(* PLC project robot6axis_ctrled, Dassault Systèmes ControlBuild 2021x HF2 *)
(* stored: creationDateTime 2021-06-01T17:00:16-01:00 *)

CONFIGURATION robot6axis_ctrled
  VAR_GLOBAL
    armOrigin AT 17 : ARRAY[1..3] OF REAL := [800.0, 400.0, 0.0];
    profileNr AT 523 : DINT := 0;
    HomeCmd AT 5 : BOOL := false;
    MoveVelCmd AT 6 : BOOL := false;
    MoveAbsCmd AT 7 : BOOL := false;
    MoveVel1ManualCmd AT 8 : BOOL := false;
    MoveVel2ManualCmd AT 9 : BOOL := false;
    MoveAbs1ManualCmd AT 10 : BOOL := false;
    MoveAbs2ManualCmd AT 11 : BOOL := false;
    StopCmd AT 12 : BOOL := false;
    MovePosition AT 22 : REAL := 0.0;
    MoveSpeed AT 23 : REAL := 100.0;
    MoveAcceleration AT 24 : REAL := 100.0;
    MoveDeceleration AT 25 : REAL := 100.0;
    offsetAxToMa AT 26 : REAL := 0.0;
    gripSyringes AT 13 : BOOL := false;
    Auto AT 14 : BOOL := false;
    Manu AT 15 : BOOL := false;
    run AT 16 : BOOL := false;
    armExtrem AT 27 : ARRAY[1..3] OF REAL := [3(0.0)];
    velX AT 32 : REAL := 0.0;
    velY AT 33 : REAL := 0.0;
    velZ AT 34 : REAL := 0.0;
    armInStop AT 17 : BOOL := false;
    masterPosition AT 35 : REAL := 0.0;
    ActualPositionAx AT 36 : REAL := 0.0;
    robot6axis_cams/profileNr AT 523 : DINT := 0;
    robot6axis_cams/HomeCmd AT 5 : BOOL := false;
    robot6axis_cams/MoveVelCmd AT 6 : BOOL := false;
    robot6axis_cams/MoveAbsCmd AT 7 : BOOL := false;
    robot6axis_cams/MoveVel1ManualCmd AT 8 : BOOL := false;
    robot6axis_cams/MoveVel2ManualCmd AT 9 : BOOL := false;
    robot6axis_cams/MoveAbs1ManualCmd AT 10 : BOOL := false;
    robot6axis_cams/MoveAbs2ManualCmd AT 11 : BOOL := false;
    robot6axis_cams/StopCmd AT 12 : BOOL := false;
    robot6axis_cams/MovePosition AT 22 : REAL := 0.0;
    robot6axis_cams/MoveSpeed AT 23 : REAL := 100.0;
    robot6axis_cams/MoveAcceleration AT 24 : REAL := 100.0;
    robot6axis_cams/MoveDeceleration AT 25 : REAL := 100.0;
    robot6axis_cams/offsetAxToMa AT 26 : REAL := 0.0;
    robot6axis_cams/name1 AT 636 : STRING(50) := 'CamAxis1_100.txt';
    robot6axis_cams/name2 AT 583 : STRING(50) := 'CamAxis2_100.txt';
    robot6axis_cams/name3 AT 530 : STRING(50) := 'CamAxis3_100.txt';
    robot6axis_cams/name4 AT 477 : STRING(50) := 'CamAxis4_100.txt';
    robot6axis_cams/name5 AT 424 : STRING(50) := 'CamAxis5_100.txt';
    robot6axis_cams/name6 AT 371 : STRING(50) := 'CamAxis6_100.txt';
    robot6axis_cams/name1_rej AT 318 : STRING(50) := 'CamAxis1_rej.txt';
    robot6axis_cams/name2_rej AT 265 : STRING(50) := 'CamAxis2_rej.txt';
    robot6axis_cams/name3_rej AT 212 : STRING(50) := 'CamAxis3_rej.txt';
    robot6axis_cams/name4_rej AT 159 : STRING(50) := 'CamAxis4_rej.txt';
    robot6axis_cams/name5_rej AT 106 : STRING(50) := 'CamAxis5_rej.txt';
    robot6axis_cams/name6_rej AT 53 : STRING(50) := 'CamAxis6_rej.txt';
    robot6axis_cams/slavePosition1 AT 158 : REAL := 0.0;
    robot6axis_cams/slavePosition2 AT 159 : REAL := 0.0;
    robot6axis_cams/slavePosition3 AT 160 : REAL := 0.0;
    robot6axis_cams/slavePosition4 AT 161 : REAL := 0.0;
    robot6axis_cams/slavePosition5 AT 162 : REAL := 0.0;
    robot6axis_cams/slavePosition6 AT 163 : REAL := 0.0;
    robot6axis_cams/ActualPositionAx AT 36 : REAL := 0.0;
    robot6axis_cams/masterPosition AT 35 : REAL := 0.0;
    robot6axis_cams/servo_kinetix2/status AT 549 : INT := 0;
    robot6axis_cams/servo_kinetix2/errorFlag AT 548 : INT := 0;
    robot6axis_cams/servo_kinetix2/ActualPositionAx1 AT 2630 : REAL := 0.0;
    robot6axis_cams/servo_kinetix2/MoveVelDone1 AT 87 : BOOL := false;
    robot6axis_cams/servo_kinetix2/ActualVelocity1 AT 2629 : REAL := 0.0;
    robot6axis_cams/servo_kinetix2/MoveAbsDone1 AT 86 : BOOL := false;
    robot6axis_cams/servo_kinetix2/HomeCmd AT 5 : BOOL := false;
    robot6axis_cams/servo_kinetix2/MoveVelCmd AT 6 : BOOL := false;
    robot6axis_cams/servo_kinetix2/MoveAbsCmd AT 7 : BOOL := false;
    robot6axis_cams/servo_kinetix2/MoveVel1ManualCmd AT 8 : BOOL := false;
    robot6axis_cams/servo_kinetix2/MoveVel2ManualCmd AT 9 : BOOL := false;
    robot6axis_cams/servo_kinetix2/MoveAbs1ManualCmd AT 10 : BOOL := false;
    robot6axis_cams/servo_kinetix2/MoveAbs2ManualCmd AT 11 : BOOL := false;
    robot6axis_cams/servo_kinetix2/StopCmd AT 12 : BOOL := false;
    robot6axis_cams/servo_kinetix2/MovePosition AT 22 : REAL := 0.0;
    robot6axis_cams/servo_kinetix2/MoveSpeed AT 23 : REAL := 100.0;
    robot6axis_cams/servo_kinetix2/MoveAcceleration AT 24 : REAL := 100.0;
    robot6axis_cams/servo_kinetix2/MoveDeceleration AT 25 : REAL := 100.0;
    robot6axis_cams/servo_kinetix2/offsetAxToMa AT 26 : REAL := 0.0;
    robot6axis_cams/servo_kinetix2/PLC_StatusReady AT 85 : BOOL := true;
    robot6axis_cams/servo_kinetix2/PLC_StatusMoved AT 84 : BOOL := false;
    robot6axis_cams/servo_kinetix2/PLC_StatusStand AT 83 : BOOL := false;
    robot6axis_cams/servo_kinetix2/PLC_ActualPositionAx AT 2628 : REAL := 0.0;
    robot6axis_cams/servo_kinetix2/PLC_ActualPositionMa AT 2627 : REAL := 0.0;
    robot6axis_cams/servo_kinetix2/PLC_ActualVelocity AT 2626 : REAL := 0.0;
    robot6axis_cams/servo_kinetix2/physicalPosInit AT 2625 : REAL := 0.0;
    robot6axis_cams/servo_kinetix2/MAX_SPEED AT 2624 : REAL(0.0..3.4e+038) := 30.0;
    robot6axis_cams/servo_kinetix2/MAX_ACCEL AT 2623 : REAL(0.0..3.4e+038) := 1500.0;
    robot6axis_cams/servo_kinetix2/MAX_DECEL AT 2622 : REAL(0.0..3.4e+038) := 1500.0;
    robot6axis_cams/servo_kinetix2/MODULO_LENGTH AT 2621 : REAL := 0.0;
    robot6axis_cams/servo_kinetix2/StatusReady AT 82 : BOOL := true;
    robot6axis_cams/servo_kinetix2/StatusMoved AT 81 : BOOL := false;
    robot6axis_cams/servo_kinetix2/StatusStand AT 80 : BOOL := false;
    robot6axis_cams/servo_kinetix2/ActualPositionAx AT 36 : REAL := 0.0;
    robot6axis_cams/servo_kinetix2/ActualPositionMa AT 2620 : REAL := 0.0;
    robot6axis_cams/servo_kinetix2/ActualVelocity AT 2619 : REAL := 0.0;
    robot6axis_cams/servo_kinetix2/MaximumVelocity AT 2618 : REAL := 0.0;
    robot6axis_cams/servo_kinetix2/StatusPosIncrease AT 79 : BOOL := false;
    robot6axis_cams/servo_kinetix2/StatusPosDecrease AT 78 : BOOL := false;
    robot6axis_cams/servo_kinetix2/displayJauge AT 2617 : REAL := 0.0;
    robot6axis_cams/servo_kinetix2/servo_mode/PLC_StatusReady AT 85 : BOOL := true;
    robot6axis_cams/servo_kinetix2/servo_mode/PLC_StatusMoved AT 84 : BOOL := false;
    robot6axis_cams/servo_kinetix2/servo_mode/PLC_StatusStand AT 83 : BOOL := false;
    robot6axis_cams/servo_kinetix2/servo_mode/PLC_ActualPositionAx AT 2628 : REAL := 0.0;
    robot6axis_cams/servo_kinetix2/servo_mode/PLC_ActualPositionMa AT 2627 : REAL := 0.0;
    robot6axis_cams/servo_kinetix2/servo_mode/PLC_ActualVelocity AT 2626 : REAL := 0.0;
    robot6axis_cams/servo_kinetix2/servo_mode/StatusReady AT 88 : BOOL := true;
    robot6axis_cams/servo_kinetix2/servo_mode/StatusMoved AT 89 : BOOL := false;
    robot6axis_cams/servo_kinetix2/servo_mode/StatusStand AT 90 : BOOL := false;
    robot6axis_cams/servo_kinetix2/servo_mode/ActualPositionMa AT 5079 : REAL := 0.0;
    robot6axis_cams/servo_kinetix2/servo_mode/ActualVelocity AT 5080 : REAL := 0.0;
    robot6axis_cams/servo_kinetix2/servo_mode/MaximumVelocity AT 5081 : REAL := 0.0;
    robot6axis_cams/servo_kinetix2/servo_mode/physicalPosInit AT 2625 : REAL := 0.0;
    robot6axis_cams/servo_kinetix2/servo_mode/ActualPositionAx AT 2630 : REAL := 0.0;
    robot6axis_cams/servo_kinetix2/servo_mode/StatusReady_o AT 82 : BOOL := true;
    robot6axis_cams/servo_kinetix2/servo_mode/StatusMoved_o AT 81 : BOOL := false;
    robot6axis_cams/servo_kinetix2/servo_mode/StatusStand_o AT 80 : BOOL := false;
    robot6axis_cams/servo_kinetix2/servo_mode/ActualPositionAx_o AT 36 : REAL := 0.0;
    robot6axis_cams/servo_kinetix2/servo_mode/ActualPositionMa_o AT 2620 : REAL := 0.0;
    robot6axis_cams/servo_kinetix2/servo_mode/ActualVelocity_o AT 2619 : REAL := 0.0;
    robot6axis_cams/servo_kinetix2/servo_mode/MaximumVelocity_o AT 2618 : REAL := 0.0;
    robot6axis_cams/servo_kinetix2/servo_mode/StatusPosIncrease_o AT 79 : BOOL := false;
    robot6axis_cams/servo_kinetix2/servo_mode/StatusPosDecrease_o AT 78 : BOOL := false;
    robot6axis_cams/servo_kinetix2/servo_mode/displayJauge_o AT 2617 : REAL := 0.0;
    robot6axis_cams/servo_kinetix2/servo_mode/PLCMode AT 95 : BOOL := false;
    robot6axis_cams/servo_kinetix2/servo_mode/PLCMode1 AT 96 : BOOL := false;
    robot6axis_cams/servo_kinetix2/servo_mode/initDone AT 97 : BOOL := false;
    robot6axis_cams/servo_kinetix2/servo_mode/displayPosMin AT 5084 : REAL := 0.0;
    robot6axis_cams/servo_kinetix2/servo_mode/displayPosMax AT 5085 : REAL := 0.0;
    robot6axis_cams/servo_kinetix2/servo_mode/PLC_ActualPositionAx1 AT 5086 : REAL := 0.0;
    robot6axis_cams/servo_kinetix2/servo_mode/PLC_ActualVelocity1 AT 5087 : REAL := 0.0;
    robot6axis_cams/servo_kinetix2/servo_mode/ActualPositionAx1 AT 5088 : REAL := 0.0;
    robot6axis_cams/servo_kinetix2/servo_mode/ActualVelocity1 AT 5089 : REAL := 0.0;
    robot6axis_cams/servo_kinetix2/servo_mode/offsetAxToMa AT 5090 : REAL := 0.0;
    robot6axis_cams/servo_kinetix2/servo_mode/offsetAxToMa1 AT 5091 : REAL := 0.0;
    robot6axis_cams/servo_kinetix2/servo_mode/ActualPositionMa_o1 AT 5092 : REAL := 0.0;
    robot6axis_cams/servo_kinetix2/servo_control/HomeCmd AT 5 : BOOL := false;
    robot6axis_cams/servo_kinetix2/servo_control/MoveVelCmd AT 6 : BOOL := false;
    robot6axis_cams/servo_kinetix2/servo_control/MoveAbsCmd AT 7 : BOOL := false;
    robot6axis_cams/servo_kinetix2/servo_control/MoveVel1ManualCmd AT 8 : BOOL := false;
    robot6axis_cams/servo_kinetix2/servo_control/MoveVel2ManualCmd AT 9 : BOOL := false;
    robot6axis_cams/servo_kinetix2/servo_control/MoveAbs1ManualCmd AT 10 : BOOL := false;
    robot6axis_cams/servo_kinetix2/servo_control/MoveAbs2ManualCmd AT 11 : BOOL := false;
    robot6axis_cams/servo_kinetix2/servo_control/StopCmd AT 12 : BOOL := false;
    robot6axis_cams/servo_kinetix2/servo_control/MovePosition AT 22 : REAL := 0.0;
    robot6axis_cams/servo_kinetix2/servo_control/MoveSpeed AT 23 : REAL := 100.0;
    robot6axis_cams/servo_kinetix2/servo_control/MoveAcceleration AT 24 : REAL := 100.0;
    robot6axis_cams/servo_kinetix2/servo_control/MoveDeceleration AT 25 : REAL := 100.0;
    robot6axis_cams/servo_kinetix2/servo_control/offsetAxToMa AT 26 : REAL := 0.0;
    robot6axis_cams/servo_kinetix2/servo_control/physicalPosInit AT 2625 : REAL := 0.0;
    robot6axis_cams/servo_kinetix2/servo_control/MAX_SPEED AT 2624 : REAL(0.0..3.4e+038) := 30.0;
    robot6axis_cams/servo_kinetix2/servo_control/status AT 549 : INT := 0;
    robot6axis_cams/servo_kinetix2/servo_control/errorFlag AT 548 : INT := 0;
    robot6axis_cams/servo_kinetix2/servo_control/IOActualPositionAx AT 2630 : REAL := 0.0;
    robot6axis_cams/servo_kinetix2/servo_control/IOVelDone AT 87 : BOOL := false;
    robot6axis_cams/servo_kinetix2/servo_control/IOAbsDone AT 86 : BOOL := false;
    robot6axis_cams/servo_kinetix2/servo_control/IOActualVelocity AT 2629 : REAL := 0.0;
    robot6axis_cams/servo_kinetix2/servo_control/OperationMode AT 574 : INT := 0;
    robot6axis_cams/servo_kinetix2/servo_control/StatusReady AT 88 : BOOL := true;
    robot6axis_cams/servo_kinetix2/servo_control/StatusMove AT 89 : BOOL := false;
    robot6axis_cams/servo_kinetix2/servo_control/StatusStand AT 90 : BOOL := false;
    robot6axis_cams/servo_kinetix2/servo_control/ActualPositionMa AT 5079 : REAL := 0.0;
    robot6axis_cams/servo_kinetix2/servo_control/ActualVelocity AT 5080 : REAL := 0.0;
    robot6axis_cams/servo_kinetix2/servo_control/MaximumVelocity AT 5081 : REAL := 0.0;
    robot6axis_cams/servo_kinetix2/servo_control/VelEnabled AT 91 : BOOL := false;
    robot6axis_cams/servo_kinetix2/servo_control/VelCmd AT 92 : BOOL := false;
    robot6axis_cams/servo_kinetix2/servo_control/PosEnabled AT 93 : BOOL := false;
    robot6axis_cams/servo_kinetix2/servo_control/PosCmd AT 94 : BOOL := false;
    robot6axis_cams/servo_kinetix2/servo_control/Position AT 5083 : REAL := 0.0;
    robot6axis_cams/servo_kinetix2/servo_control/Speed AT 5082 : REAL := 0.0;
    robot6axis_cams/servo_kinetix2/servo_control/ManualMode AT 575 : INT := 0;
    robot6axis_cams/servo_kinetix2/servo_control/initDone AT 98 : BOOL := false;
    robot6axis_cams/servo_kinetix2/servo_control/ActualPositionMa1 AT 5093 : REAL := 0.0;
    robot6axis_cams/servo_kinetix2/servo_control/offsetAxToMa1 AT 5094 : REAL := 0.0;
    robot6axis_cams/servo_kinetix2/servo_control/HOME_POSITION AT 5095 : REAL := 100.0;
    robot6axis_cams/servo_kinetix2/servo_control/MANUAL_POSITION1 AT 5096 : REAL := 0.0;
    robot6axis_cams/servo_kinetix2/servo_control/MANUAL_POSITION2 AT 5097 : REAL := 150.0;
    robot6axis_cams/servo_kinetix2/servo_control/MANUAL_SPEED1 AT 5098 : REAL := -100.0;
    robot6axis_cams/servo_kinetix2/servo_control/MANUAL_SPEED2 AT 5099 : REAL := 100.0;
    robot6axis_cams/servo_kinetix2/servo_control/MANUAL_SPEED AT 5100 : REAL := 100.0;
    robot6axis_cams/servo_kinetix2/servo_velocity/MoveVelEnable AT 91 : BOOL := false;
    robot6axis_cams/servo_kinetix2/servo_velocity/MoveVelStart AT 92 : BOOL := false;
    robot6axis_cams/servo_kinetix2/servo_velocity/MoveSpeed AT 5082 : REAL := 0.0;
    robot6axis_cams/servo_kinetix2/servo_velocity/MoveAcceleration AT 24 : REAL := 100.0;
    robot6axis_cams/servo_kinetix2/servo_velocity/MoveDeceleration AT 25 : REAL := 100.0;
    robot6axis_cams/servo_kinetix2/servo_velocity/MAX_SPEED AT 2624 : REAL(0.0..3.4e+038) := 30.0;
    robot6axis_cams/servo_kinetix2/servo_velocity/MAX_ACCEL AT 2623 : REAL(0.0..3.4e+038) := 1500.0;
    robot6axis_cams/servo_kinetix2/servo_velocity/MAX_DECEL AT 2622 : REAL(0.0..3.4e+038) := 1500.0;
    robot6axis_cams/servo_kinetix2/servo_velocity/MODULO_LENGTH AT 2621 : REAL := 0.0;
    robot6axis_cams/servo_kinetix2/servo_velocity/status AT 549 : INT := 0;
    robot6axis_cams/servo_kinetix2/servo_velocity/errorFlag AT 548 : INT := 0;
    robot6axis_cams/servo_kinetix2/servo_velocity/MoveVelDone AT 87 : BOOL := false;
    robot6axis_cams/servo_kinetix2/servo_velocity/ActualPositionAx AT 2630 : REAL := 0.0;
    robot6axis_cams/servo_kinetix2/servo_velocity/ActualVelocity AT 2629 : REAL := 0.0;
    robot6axis_cams/servo_kinetix2/servo_velocity/firstStep AT 99 : BOOL := true;
    robot6axis_cams/servo_kinetix2/servo_velocity/stepDone AT 100 : BOOL := false;
    robot6axis_cams/servo_kinetix2/servo_velocity/currentTime AT 5101 : REAL := 0.0;
    robot6axis_cams/servo_kinetix2/servo_velocity/MoveSpeed1 AT 5102 : REAL := 0.0;
    robot6axis_cams/servo_kinetix2/servo_velocity/acceleration AT 5103 : REAL := 0.0;
    robot6axis_cams/servo_kinetix2/servo_velocity/deceleration AT 5104 : REAL := 0.0;
    robot6axis_cams/servo_kinetix2/servo_velocity/orderSpeed AT 5105 : REAL := 0.0;
    robot6axis_cams/servo_kinetix2/servo_velocity/endChangeSpeed AT 5106 : REAL := 0.0;
    robot6axis_cams/servo_kinetix2/servo_velocity/accelDecelChangeSpeed AT 5107 : REAL := 0.0;
    robot6axis_cams/servo_kinetix2/servo_velocity/ActualVelocity1 AT 5108 : REAL := 0.0;
    robot6axis_cams/servo_kinetix2/servo_velocity/speedChanged AT 101 : BOOL := false;
    robot6axis_cams/servo_kinetix2/servo_position/MoveAbsEnable AT 93 : BOOL := false;
    robot6axis_cams/servo_kinetix2/servo_position/MoveAbsStart AT 94 : BOOL := false;
    robot6axis_cams/servo_kinetix2/servo_position/MovePosition AT 5083 : REAL := 0.0;
    robot6axis_cams/servo_kinetix2/servo_position/MoveSpeed AT 5082 : REAL := 0.0;
    robot6axis_cams/servo_kinetix2/servo_position/MoveAcceleration AT 24 : REAL := 100.0;
    robot6axis_cams/servo_kinetix2/servo_position/MoveDeceleration AT 25 : REAL := 100.0;
    robot6axis_cams/servo_kinetix2/servo_position/MAX_SPEED AT 2624 : REAL(0.0..3.4e+038) := 30.0;
    robot6axis_cams/servo_kinetix2/servo_position/MAX_ACCEL AT 2623 : REAL(0.0..3.4e+038) := 1500.0;
    robot6axis_cams/servo_kinetix2/servo_position/MAX_DECEL AT 2622 : REAL(0.0..3.4e+038) := 1500.0;
    robot6axis_cams/servo_kinetix2/servo_position/MODULO_LENGTH AT 2621 : REAL := 0.0;
    robot6axis_cams/servo_kinetix2/servo_position/status AT 549 : INT := 0;
    robot6axis_cams/servo_kinetix2/servo_position/errorFlag AT 548 : INT := 0;
    robot6axis_cams/servo_kinetix2/servo_position/MoveAbsDone AT 86 : BOOL := false;
    robot6axis_cams/servo_kinetix2/servo_position/ActualPositionAx AT 2630 : REAL := 0.0;
    robot6axis_cams/servo_kinetix2/servo_position/ActualVelocity AT 2629 : REAL := 0.0;
    robot6axis_cams/servo_kinetix2/servo_position/firstStep AT 102 : BOOL := true;
    robot6axis_cams/servo_kinetix2/servo_position/stepDone AT 103 : BOOL := false;
    robot6axis_cams/servo_kinetix2/servo_position/timeToStop AT 5109 : REAL := 0.0;
    robot6axis_cams/servo_kinetix2/servo_position/distanceToStop AT 5110 : REAL := 0.0;
    robot6axis_cams/servo_kinetix2/servo_position/distance AT 5111 : REAL := 0.0;
    robot6axis_cams/servo_kinetix2/servo_position/currentTime AT 5112 : REAL := 0.0;
    robot6axis_cams/servo_kinetix2/servo_position/currentSpeed1 AT 5113 : REAL := 0.0;
    robot6axis_cams/servo_kinetix2/servo_position/targetPosition AT 5114 : REAL := 0.0;
    robot6axis_cams/servo_kinetix2/servo_position/ActualPositionAx1 AT 5115 : REAL := 0.0;
    robot6axis_cams/servo_kinetix2/servo_position/acceleration AT 5116 : REAL := 0.0;
    robot6axis_cams/servo_kinetix2/servo_position/deceleration AT 5117 : REAL := 0.0;
    robot6axis_cams/servo_kinetix2/servo_position/orderSpeed AT 5118 : REAL := 0.0;
    robot6axis_cams/servo_kinetix2/servo_position/moveDirection AT 5119 : REAL := 0.0;
    robot6axis_cams/servo_kinetix2/servo_position/moveDirection1 AT 5120 : REAL := 0.0;
    robot6axis_cams/servo_kinetix2/servo_position/endChangeSpeed AT 5121 : REAL := 0.0;
    robot6axis_cams/servo_kinetix2/servo_position/ActualVelocity1 AT 5122 : REAL := 0.0;
    robot6axis_cams/cam_profile1/name AT 636 : STRING(50) := 'CamAxis1_100.txt';
    robot6axis_cams/cam_profile1/nbPoints AT 550 : INT := 0;
    robot6axis_cams/cam_profile1/MasterPoints AT 2631 : ARRAY[1..100] OF REAL := [100(0.0)];
    robot6axis_cams/cam_profile1/SlavePoints AT 2733 : ARRAY[1..100] OF REAL := [100(0.0)];
    robot6axis_cams/cam_profile1/pointer AT 551 : DINT := 0;
    robot6axis_cams/cam_profile1/initialized AT 104 : BOOL := false;
    robot6axis_cams/cam_profile1/pFile AT 576 : DINT := 0;
    robot6axis_cams/cam_profile1/fault_reading AT 105 : BOOL := false;
    robot6axis_cams/cam_profile1/fault_openning AT 106 : BOOL := false;
    robot6axis_cams/cam_profile1/complete_path AT 689 : STRING(254) := '';
    robot6axis_cams/cam_profile7/name AT 318 : STRING(50) := 'CamAxis1_rej.txt';
    robot6axis_cams/cam_profile7/nbPoints AT 552 : INT := 0;
    robot6axis_cams/cam_profile7/MasterPoints AT 2835 : ARRAY[1..100] OF REAL := [100(0.0)];
    robot6axis_cams/cam_profile7/SlavePoints AT 2937 : ARRAY[1..100] OF REAL := [100(0.0)];
    robot6axis_cams/cam_profile7/pointer AT 553 : DINT := 0;
    robot6axis_cams/cam_profile7/initialized AT 107 : BOOL := false;
    robot6axis_cams/cam_profile7/pFile AT 577 : DINT := 0;
    robot6axis_cams/cam_profile7/fault_reading AT 108 : BOOL := false;
    robot6axis_cams/cam_profile7/fault_openning AT 109 : BOOL := false;
    robot6axis_cams/cam_profile7/complete_path AT 946 : STRING(254) := '';
    robot6axis_cams/cam_computation1/profileNr AT 523 : DINT := 0;
    robot6axis_cams/cam_computation1/MasterPositionIn AT 36 : REAL := 0.0;
    robot6axis_cams/cam_computation1/nbPoints0 AT 550 : INT := 0;
    robot6axis_cams/cam_computation1/MasterPoints0 AT 2631 : ARRAY[1..100] OF REAL := [100(0.0)];
    robot6axis_cams/cam_computation1/SlavePoints0 AT 2733 : ARRAY[1..100] OF REAL := [100(0.0)];
    robot6axis_cams/cam_computation1/pointer0 AT 551 : DINT := 0;
    robot6axis_cams/cam_computation1/nbPoints1 AT 552 : INT := 0;
    robot6axis_cams/cam_computation1/MasterPoints1 AT 2835 : ARRAY[1..100] OF REAL := [100(0.0)];
    robot6axis_cams/cam_computation1/SlavePoints1 AT 2937 : ARRAY[1..100] OF REAL := [100(0.0)];
    robot6axis_cams/cam_computation1/pointer1 AT 553 : DINT := 0;
    robot6axis_cams/cam_computation1/nbPoints2 AT 547 : INT := 0;
    robot6axis_cams/cam_computation1/MasterPoints2 AT 2515 : ARRAY[1..100] OF REAL := [100(0.0)];
    robot6axis_cams/cam_computation1/SlavePoints2 AT 2413 : ARRAY[1..100] OF REAL := [100(0.0)];
    robot6axis_cams/cam_computation1/pointer2 AT 546 : DINT := 0;
    robot6axis_cams/cam_computation1/nbPoints3 AT 545 : INT := 0;
    robot6axis_cams/cam_computation1/MasterPoints3 AT 2311 : ARRAY[1..100] OF REAL := [100(0.0)];
    robot6axis_cams/cam_computation1/SlavePoints3 AT 2209 : ARRAY[1..100] OF REAL := [100(0.0)];
    robot6axis_cams/cam_computation1/pointer3 AT 544 : DINT := 0;
    robot6axis_cams/cam_computation1/slavePosition AT 158 : REAL := 0.0;
    robot6axis_cams/cam_computation1/masterPosition AT 35 : REAL := 0.0;
    robot6axis_cams/cam_computation1/i AT 578 : INT := 0;
    robot6axis_cams/cam_computation1/modulo AT 5123 : REAL := 0.0;
    robot6axis_cams/cam_computation1/divider AT 579 : INT := 0;
    robot6axis_cams/cam_computation1/faultProfileNr AT 110 : BOOL := false;
    robot6axis_cams/cam_computation1/faultMasterPositionOOB AT 111 : BOOL := false;
    robot6axis_cams/cam_computation1/faultLinComputation AT 112 : BOOL := false;
    robot6axis_cams/cam_computation1/nbPoints AT 580 : INT := 0;
    robot6axis_cams/cam_computation1/MasterPoints AT 5124 : ARRAY[1..100] OF REAL := [100(0.0)];
    robot6axis_cams/cam_computation1/SlavePoints AT 5226 : ARRAY[1..100] OF REAL := [100(0.0)];
    robot6axis_cams/cam_computation1/found AT 113 : BOOL := false;
    robot6axis_cams/cam_computation1/index AT 581 : INT := 0;
    robot6axis_cams/cam_computation1/linDenom AT 5328 : REAL := 0.0;
    robot6axis_cams/cam_computation1/linNum AT 5329 : REAL := 0.0;
    robot6axis_cams/cam_computation1/linA AT 5330 : REAL := 0.0;
    robot6axis_cams/cam_computation1/linB AT 5331 : REAL := 0.0;
    robot6axis_cams/cam_computation1/FACTOR AT 5332 : REAL := 1.0;
    robot6axis_cams/cam_profile2/name AT 583 : STRING(50) := 'CamAxis2_100.txt';
    robot6axis_cams/cam_profile2/nbPoints AT 554 : INT := 0;
    robot6axis_cams/cam_profile2/MasterPoints AT 3039 : ARRAY[1..100] OF REAL := [100(0.0)];
    robot6axis_cams/cam_profile2/SlavePoints AT 3141 : ARRAY[1..100] OF REAL := [100(0.0)];
    robot6axis_cams/cam_profile2/pointer AT 555 : DINT := 0;
    robot6axis_cams/cam_profile2/initialized AT 114 : BOOL := false;
    robot6axis_cams/cam_profile2/pFile AT 582 : DINT := 0;
    robot6axis_cams/cam_profile2/fault_reading AT 115 : BOOL := false;
    robot6axis_cams/cam_profile2/fault_openning AT 116 : BOOL := false;
    robot6axis_cams/cam_profile2/complete_path AT 1203 : STRING(254) := '';
    robot6axis_cams/cam_profile8/name AT 265 : STRING(50) := 'CamAxis2_rej.txt';
    robot6axis_cams/cam_profile8/nbPoints AT 556 : INT := 0;
    robot6axis_cams/cam_profile8/MasterPoints AT 3243 : ARRAY[1..100] OF REAL := [100(0.0)];
    robot6axis_cams/cam_profile8/SlavePoints AT 3345 : ARRAY[1..100] OF REAL := [100(0.0)];
    robot6axis_cams/cam_profile8/pointer AT 557 : DINT := 0;
    robot6axis_cams/cam_profile8/initialized AT 117 : BOOL := false;
    robot6axis_cams/cam_profile8/pFile AT 583 : DINT := 0;
    robot6axis_cams/cam_profile8/fault_reading AT 118 : BOOL := false;
    robot6axis_cams/cam_profile8/fault_openning AT 119 : BOOL := false;
    robot6axis_cams/cam_profile8/complete_path AT 1460 : STRING(254) := '';
    robot6axis_cams/cam_computation2/profileNr AT 523 : DINT := 0;
    robot6axis_cams/cam_computation2/MasterPositionIn AT 36 : REAL := 0.0;
    robot6axis_cams/cam_computation2/nbPoints0 AT 554 : INT := 0;
    robot6axis_cams/cam_computation2/MasterPoints0 AT 3039 : ARRAY[1..100] OF REAL := [100(0.0)];
    robot6axis_cams/cam_computation2/SlavePoints0 AT 3141 : ARRAY[1..100] OF REAL := [100(0.0)];
    robot6axis_cams/cam_computation2/pointer0 AT 555 : DINT := 0;
    robot6axis_cams/cam_computation2/nbPoints1 AT 556 : INT := 0;
    robot6axis_cams/cam_computation2/MasterPoints1 AT 3243 : ARRAY[1..100] OF REAL := [100(0.0)];
    robot6axis_cams/cam_computation2/SlavePoints1 AT 3345 : ARRAY[1..100] OF REAL := [100(0.0)];
    robot6axis_cams/cam_computation2/pointer1 AT 557 : DINT := 0;
    robot6axis_cams/cam_computation2/nbPoints2 AT 543 : INT := 0;
    robot6axis_cams/cam_computation2/MasterPoints2 AT 2107 : ARRAY[1..100] OF REAL := [100(0.0)];
    robot6axis_cams/cam_computation2/SlavePoints2 AT 2005 : ARRAY[1..100] OF REAL := [100(0.0)];
    robot6axis_cams/cam_computation2/pointer2 AT 542 : DINT := 0;
    robot6axis_cams/cam_computation2/nbPoints3 AT 541 : INT := 0;
    robot6axis_cams/cam_computation2/MasterPoints3 AT 1903 : ARRAY[1..100] OF REAL := [100(0.0)];
    robot6axis_cams/cam_computation2/SlavePoints3 AT 1801 : ARRAY[1..100] OF REAL := [100(0.0)];
    robot6axis_cams/cam_computation2/pointer3 AT 540 : DINT := 0;
    robot6axis_cams/cam_computation2/slavePosition AT 159 : REAL := 0.0;
    robot6axis_cams/cam_computation2/masterPosition AT 1800 : REAL := 0.0;
    robot6axis_cams/cam_computation2/i AT 584 : INT := 0;
    robot6axis_cams/cam_computation2/modulo AT 5333 : REAL := 0.0;
    robot6axis_cams/cam_computation2/divider AT 585 : INT := 0;
    robot6axis_cams/cam_computation2/faultProfileNr AT 120 : BOOL := false;
    robot6axis_cams/cam_computation2/faultMasterPositionOOB AT 121 : BOOL := false;
    robot6axis_cams/cam_computation2/faultLinComputation AT 122 : BOOL := false;
    robot6axis_cams/cam_computation2/nbPoints AT 586 : INT := 0;
    robot6axis_cams/cam_computation2/MasterPoints AT 5334 : ARRAY[1..100] OF REAL := [100(0.0)];
    robot6axis_cams/cam_computation2/SlavePoints AT 5436 : ARRAY[1..100] OF REAL := [100(0.0)];
    robot6axis_cams/cam_computation2/found AT 123 : BOOL := false;
    robot6axis_cams/cam_computation2/index AT 587 : INT := 0;
    robot6axis_cams/cam_computation2/linDenom AT 5538 : REAL := 0.0;
    robot6axis_cams/cam_computation2/linNum AT 5539 : REAL := 0.0;
    robot6axis_cams/cam_computation2/linA AT 5540 : REAL := 0.0;
    robot6axis_cams/cam_computation2/linB AT 5541 : REAL := 0.0;
    robot6axis_cams/cam_computation2/FACTOR AT 5542 : REAL := 1.0;
    robot6axis_cams/cam_profile3/name AT 530 : STRING(50) := 'CamAxis3_100.txt';
    robot6axis_cams/cam_profile3/nbPoints AT 558 : INT := 0;
    robot6axis_cams/cam_profile3/MasterPoints AT 3447 : ARRAY[1..100] OF REAL := [100(0.0)];
    robot6axis_cams/cam_profile3/SlavePoints AT 3549 : ARRAY[1..100] OF REAL := [100(0.0)];
    robot6axis_cams/cam_profile3/pointer AT 559 : DINT := 0;
    robot6axis_cams/cam_profile3/initialized AT 124 : BOOL := false;
    robot6axis_cams/cam_profile3/pFile AT 588 : DINT := 0;
    robot6axis_cams/cam_profile3/fault_reading AT 125 : BOOL := false;
    robot6axis_cams/cam_profile3/fault_openning AT 126 : BOOL := false;
    robot6axis_cams/cam_profile3/complete_path AT 1717 : STRING(254) := '';
    robot6axis_cams/cam_profile9/name AT 212 : STRING(50) := 'CamAxis3_rej.txt';
    robot6axis_cams/cam_profile9/nbPoints AT 560 : INT := 0;
    robot6axis_cams/cam_profile9/MasterPoints AT 3651 : ARRAY[1..100] OF REAL := [100(0.0)];
    robot6axis_cams/cam_profile9/SlavePoints AT 3753 : ARRAY[1..100] OF REAL := [100(0.0)];
    robot6axis_cams/cam_profile9/pointer AT 561 : DINT := 0;
    robot6axis_cams/cam_profile9/initialized AT 127 : BOOL := false;
    robot6axis_cams/cam_profile9/pFile AT 589 : DINT := 0;
    robot6axis_cams/cam_profile9/fault_reading AT 128 : BOOL := false;
    robot6axis_cams/cam_profile9/fault_openning AT 129 : BOOL := false;
    robot6axis_cams/cam_profile9/complete_path AT 1974 : STRING(254) := '';
    robot6axis_cams/cam_computation3/profileNr AT 523 : DINT := 0;
    robot6axis_cams/cam_computation3/MasterPositionIn AT 36 : REAL := 0.0;
    robot6axis_cams/cam_computation3/nbPoints0 AT 558 : INT := 0;
    robot6axis_cams/cam_computation3/MasterPoints0 AT 3447 : ARRAY[1..100] OF REAL := [100(0.0)];
    robot6axis_cams/cam_computation3/SlavePoints0 AT 3549 : ARRAY[1..100] OF REAL := [100(0.0)];
    robot6axis_cams/cam_computation3/pointer0 AT 559 : DINT := 0;
    robot6axis_cams/cam_computation3/nbPoints1 AT 560 : INT := 0;
    robot6axis_cams/cam_computation3/MasterPoints1 AT 3651 : ARRAY[1..100] OF REAL := [100(0.0)];
    robot6axis_cams/cam_computation3/SlavePoints1 AT 3753 : ARRAY[1..100] OF REAL := [100(0.0)];
    robot6axis_cams/cam_computation3/pointer1 AT 561 : DINT := 0;
    robot6axis_cams/cam_computation3/nbPoints2 AT 539 : INT := 0;
    robot6axis_cams/cam_computation3/MasterPoints2 AT 1698 : ARRAY[1..100] OF REAL := [100(0.0)];
    robot6axis_cams/cam_computation3/SlavePoints2 AT 1596 : ARRAY[1..100] OF REAL := [100(0.0)];
    robot6axis_cams/cam_computation3/pointer2 AT 538 : DINT := 0;
    robot6axis_cams/cam_computation3/nbPoints3 AT 537 : INT := 0;
    robot6axis_cams/cam_computation3/MasterPoints3 AT 1494 : ARRAY[1..100] OF REAL := [100(0.0)];
    robot6axis_cams/cam_computation3/SlavePoints3 AT 1392 : ARRAY[1..100] OF REAL := [100(0.0)];
    robot6axis_cams/cam_computation3/pointer3 AT 536 : DINT := 0;
    robot6axis_cams/cam_computation3/slavePosition AT 160 : REAL := 0.0;
    robot6axis_cams/cam_computation3/masterPosition AT 1391 : REAL := 0.0;
    robot6axis_cams/cam_computation3/i AT 590 : INT := 0;
    robot6axis_cams/cam_computation3/modulo AT 5543 : REAL := 0.0;
    robot6axis_cams/cam_computation3/divider AT 591 : INT := 0;
    robot6axis_cams/cam_computation3/faultProfileNr AT 130 : BOOL := false;
    robot6axis_cams/cam_computation3/faultMasterPositionOOB AT 131 : BOOL := false;
    robot6axis_cams/cam_computation3/faultLinComputation AT 132 : BOOL := false;
    robot6axis_cams/cam_computation3/nbPoints AT 592 : INT := 0;
    robot6axis_cams/cam_computation3/MasterPoints AT 5544 : ARRAY[1..100] OF REAL := [100(0.0)];
    robot6axis_cams/cam_computation3/SlavePoints AT 5646 : ARRAY[1..100] OF REAL := [100(0.0)];
    robot6axis_cams/cam_computation3/found AT 133 : BOOL := false;
    robot6axis_cams/cam_computation3/index AT 593 : INT := 0;
    robot6axis_cams/cam_computation3/linDenom AT 5748 : REAL := 0.0;
    robot6axis_cams/cam_computation3/linNum AT 5749 : REAL := 0.0;
    robot6axis_cams/cam_computation3/linA AT 5750 : REAL := 0.0;
    robot6axis_cams/cam_computation3/linB AT 5751 : REAL := 0.0;
    robot6axis_cams/cam_computation3/FACTOR AT 5752 : REAL := 1.0;
    robot6axis_cams/cam_profile4/name AT 477 : STRING(50) := 'CamAxis4_100.txt';
    robot6axis_cams/cam_profile4/nbPoints AT 562 : INT := 0;
    robot6axis_cams/cam_profile4/MasterPoints AT 3855 : ARRAY[1..100] OF REAL := [100(0.0)];
    robot6axis_cams/cam_profile4/SlavePoints AT 3957 : ARRAY[1..100] OF REAL := [100(0.0)];
    robot6axis_cams/cam_profile4/pointer AT 563 : DINT := 0;
    robot6axis_cams/cam_profile4/initialized AT 134 : BOOL := false;
    robot6axis_cams/cam_profile4/pFile AT 594 : DINT := 0;
    robot6axis_cams/cam_profile4/fault_reading AT 135 : BOOL := false;
    robot6axis_cams/cam_profile4/fault_openning AT 136 : BOOL := false;
    robot6axis_cams/cam_profile4/complete_path AT 2231 : STRING(254) := '';
    robot6axis_cams/cam_profile10/name AT 159 : STRING(50) := 'CamAxis4_rej.txt';
    robot6axis_cams/cam_profile10/nbPoints AT 564 : INT := 0;
    robot6axis_cams/cam_profile10/MasterPoints AT 4059 : ARRAY[1..100] OF REAL := [100(0.0)];
    robot6axis_cams/cam_profile10/SlavePoints AT 4161 : ARRAY[1..100] OF REAL := [100(0.0)];
    robot6axis_cams/cam_profile10/pointer AT 565 : DINT := 0;
    robot6axis_cams/cam_profile10/initialized AT 137 : BOOL := false;
    robot6axis_cams/cam_profile10/pFile AT 595 : DINT := 0;
    robot6axis_cams/cam_profile10/fault_reading AT 138 : BOOL := false;
    robot6axis_cams/cam_profile10/fault_openning AT 139 : BOOL := false;
    robot6axis_cams/cam_profile10/complete_path AT 2488 : STRING(254) := '';
    robot6axis_cams/cam_computation4/profileNr AT 523 : DINT := 0;
    robot6axis_cams/cam_computation4/MasterPositionIn AT 36 : REAL := 0.0;
    robot6axis_cams/cam_computation4/nbPoints0 AT 562 : INT := 0;
    robot6axis_cams/cam_computation4/MasterPoints0 AT 3855 : ARRAY[1..100] OF REAL := [100(0.0)];
    robot6axis_cams/cam_computation4/SlavePoints0 AT 3957 : ARRAY[1..100] OF REAL := [100(0.0)];
    robot6axis_cams/cam_computation4/pointer0 AT 563 : DINT := 0;
    robot6axis_cams/cam_computation4/nbPoints1 AT 564 : INT := 0;
    robot6axis_cams/cam_computation4/MasterPoints1 AT 4059 : ARRAY[1..100] OF REAL := [100(0.0)];
    robot6axis_cams/cam_computation4/SlavePoints1 AT 4161 : ARRAY[1..100] OF REAL := [100(0.0)];
    robot6axis_cams/cam_computation4/pointer1 AT 565 : DINT := 0;
    robot6axis_cams/cam_computation4/nbPoints2 AT 535 : INT := 0;
    robot6axis_cams/cam_computation4/MasterPoints2 AT 1289 : ARRAY[1..100] OF REAL := [100(0.0)];
    robot6axis_cams/cam_computation4/SlavePoints2 AT 1187 : ARRAY[1..100] OF REAL := [100(0.0)];
    robot6axis_cams/cam_computation4/pointer2 AT 534 : DINT := 0;
    robot6axis_cams/cam_computation4/nbPoints3 AT 533 : INT := 0;
    robot6axis_cams/cam_computation4/MasterPoints3 AT 1085 : ARRAY[1..100] OF REAL := [100(0.0)];
    robot6axis_cams/cam_computation4/SlavePoints3 AT 983 : ARRAY[1..100] OF REAL := [100(0.0)];
    robot6axis_cams/cam_computation4/pointer3 AT 532 : DINT := 0;
    robot6axis_cams/cam_computation4/slavePosition AT 161 : REAL := 0.0;
    robot6axis_cams/cam_computation4/masterPosition AT 982 : REAL := 0.0;
    robot6axis_cams/cam_computation4/i AT 596 : INT := 0;
    robot6axis_cams/cam_computation4/modulo AT 5753 : REAL := 0.0;
    robot6axis_cams/cam_computation4/divider AT 597 : INT := 0;
    robot6axis_cams/cam_computation4/faultProfileNr AT 140 : BOOL := false;
    robot6axis_cams/cam_computation4/faultMasterPositionOOB AT 141 : BOOL := false;
    robot6axis_cams/cam_computation4/faultLinComputation AT 142 : BOOL := false;
    robot6axis_cams/cam_computation4/nbPoints AT 598 : INT := 0;
    robot6axis_cams/cam_computation4/MasterPoints AT 5754 : ARRAY[1..100] OF REAL := [100(0.0)];
    robot6axis_cams/cam_computation4/SlavePoints AT 5856 : ARRAY[1..100] OF REAL := [100(0.0)];
    robot6axis_cams/cam_computation4/found AT 143 : BOOL := false;
    robot6axis_cams/cam_computation4/index AT 599 : INT := 0;
    robot6axis_cams/cam_computation4/linDenom AT 5958 : REAL := 0.0;
    robot6axis_cams/cam_computation4/linNum AT 5959 : REAL := 0.0;
    robot6axis_cams/cam_computation4/linA AT 5960 : REAL := 0.0;
    robot6axis_cams/cam_computation4/linB AT 5961 : REAL := 0.0;
    robot6axis_cams/cam_computation4/FACTOR AT 5962 : REAL := 1.0;
    robot6axis_cams/cam_profile5/name AT 424 : STRING(50) := 'CamAxis5_100.txt';
    robot6axis_cams/cam_profile5/nbPoints AT 566 : INT := 0;
    robot6axis_cams/cam_profile5/MasterPoints AT 4263 : ARRAY[1..100] OF REAL := [100(0.0)];
    robot6axis_cams/cam_profile5/SlavePoints AT 4365 : ARRAY[1..100] OF REAL := [100(0.0)];
    robot6axis_cams/cam_profile5/pointer AT 567 : DINT := 0;
    robot6axis_cams/cam_profile5/initialized AT 144 : BOOL := false;
    robot6axis_cams/cam_profile5/pFile AT 600 : DINT := 0;
    robot6axis_cams/cam_profile5/fault_reading AT 145 : BOOL := false;
    robot6axis_cams/cam_profile5/fault_openning AT 146 : BOOL := false;
    robot6axis_cams/cam_profile5/complete_path AT 2745 : STRING(254) := '';
    robot6axis_cams/cam_profile11/name AT 106 : STRING(50) := 'CamAxis5_rej.txt';
    robot6axis_cams/cam_profile11/nbPoints AT 568 : INT := 0;
    robot6axis_cams/cam_profile11/MasterPoints AT 4467 : ARRAY[1..100] OF REAL := [100(0.0)];
    robot6axis_cams/cam_profile11/SlavePoints AT 4569 : ARRAY[1..100] OF REAL := [100(0.0)];
    robot6axis_cams/cam_profile11/pointer AT 569 : DINT := 0;
    robot6axis_cams/cam_profile11/initialized AT 147 : BOOL := false;
    robot6axis_cams/cam_profile11/pFile AT 601 : DINT := 0;
    robot6axis_cams/cam_profile11/fault_reading AT 148 : BOOL := false;
    robot6axis_cams/cam_profile11/fault_openning AT 149 : BOOL := false;
    robot6axis_cams/cam_profile11/complete_path AT 3002 : STRING(254) := '';
    robot6axis_cams/cam_computation5/profileNr AT 523 : DINT := 0;
    robot6axis_cams/cam_computation5/MasterPositionIn AT 36 : REAL := 0.0;
    robot6axis_cams/cam_computation5/nbPoints0 AT 566 : INT := 0;
    robot6axis_cams/cam_computation5/MasterPoints0 AT 4263 : ARRAY[1..100] OF REAL := [100(0.0)];
    robot6axis_cams/cam_computation5/SlavePoints0 AT 4365 : ARRAY[1..100] OF REAL := [100(0.0)];
    robot6axis_cams/cam_computation5/pointer0 AT 567 : DINT := 0;
    robot6axis_cams/cam_computation5/nbPoints1 AT 568 : INT := 0;
    robot6axis_cams/cam_computation5/MasterPoints1 AT 4467 : ARRAY[1..100] OF REAL := [100(0.0)];
    robot6axis_cams/cam_computation5/SlavePoints1 AT 4569 : ARRAY[1..100] OF REAL := [100(0.0)];
    robot6axis_cams/cam_computation5/pointer1 AT 569 : DINT := 0;
    robot6axis_cams/cam_computation5/nbPoints2 AT 531 : INT := 0;
    robot6axis_cams/cam_computation5/MasterPoints2 AT 880 : ARRAY[1..100] OF REAL := [100(0.0)];
    robot6axis_cams/cam_computation5/SlavePoints2 AT 778 : ARRAY[1..100] OF REAL := [100(0.0)];
    robot6axis_cams/cam_computation5/pointer2 AT 530 : DINT := 0;
    robot6axis_cams/cam_computation5/nbPoints3 AT 529 : INT := 0;
    robot6axis_cams/cam_computation5/MasterPoints3 AT 676 : ARRAY[1..100] OF REAL := [100(0.0)];
    robot6axis_cams/cam_computation5/SlavePoints3 AT 574 : ARRAY[1..100] OF REAL := [100(0.0)];
    robot6axis_cams/cam_computation5/pointer3 AT 528 : DINT := 0;
    robot6axis_cams/cam_computation5/slavePosition AT 162 : REAL := 0.0;
    robot6axis_cams/cam_computation5/masterPosition AT 573 : REAL := 0.0;
    robot6axis_cams/cam_computation5/i AT 602 : INT := 0;
    robot6axis_cams/cam_computation5/modulo AT 5963 : REAL := 0.0;
    robot6axis_cams/cam_computation5/divider AT 603 : INT := 0;
    robot6axis_cams/cam_computation5/faultProfileNr AT 150 : BOOL := false;
    robot6axis_cams/cam_computation5/faultMasterPositionOOB AT 151 : BOOL := false;
    robot6axis_cams/cam_computation5/faultLinComputation AT 152 : BOOL := false;
    robot6axis_cams/cam_computation5/nbPoints AT 604 : INT := 0;
    robot6axis_cams/cam_computation5/MasterPoints AT 5964 : ARRAY[1..100] OF REAL := [100(0.0)];
    robot6axis_cams/cam_computation5/SlavePoints AT 6066 : ARRAY[1..100] OF REAL := [100(0.0)];
    robot6axis_cams/cam_computation5/found AT 153 : BOOL := false;
    robot6axis_cams/cam_computation5/index AT 605 : INT := 0;
    robot6axis_cams/cam_computation5/linDenom AT 6168 : REAL := 0.0;
    robot6axis_cams/cam_computation5/linNum AT 6169 : REAL := 0.0;
    robot6axis_cams/cam_computation5/linA AT 6170 : REAL := 0.0;
    robot6axis_cams/cam_computation5/linB AT 6171 : REAL := 0.0;
    robot6axis_cams/cam_computation5/FACTOR AT 6172 : REAL := 1.0;
    robot6axis_cams/cam_profile6/name AT 371 : STRING(50) := 'CamAxis6_100.txt';
    robot6axis_cams/cam_profile6/nbPoints AT 570 : INT := 0;
    robot6axis_cams/cam_profile6/MasterPoints AT 4671 : ARRAY[1..100] OF REAL := [100(0.0)];
    robot6axis_cams/cam_profile6/SlavePoints AT 4773 : ARRAY[1..100] OF REAL := [100(0.0)];
    robot6axis_cams/cam_profile6/pointer AT 571 : DINT := 0;
    robot6axis_cams/cam_profile6/initialized AT 154 : BOOL := false;
    robot6axis_cams/cam_profile6/pFile AT 606 : DINT := 0;
    robot6axis_cams/cam_profile6/fault_reading AT 155 : BOOL := false;
    robot6axis_cams/cam_profile6/fault_openning AT 156 : BOOL := false;
    robot6axis_cams/cam_profile6/complete_path AT 3259 : STRING(254) := '';
    robot6axis_cams/cam_profile12/name AT 53 : STRING(50) := 'CamAxis6_rej.txt';
    robot6axis_cams/cam_profile12/nbPoints AT 572 : INT := 0;
    robot6axis_cams/cam_profile12/MasterPoints AT 4875 : ARRAY[1..100] OF REAL := [100(0.0)];
    robot6axis_cams/cam_profile12/SlavePoints AT 4977 : ARRAY[1..100] OF REAL := [100(0.0)];
    robot6axis_cams/cam_profile12/pointer AT 573 : DINT := 0;
    robot6axis_cams/cam_profile12/initialized AT 157 : BOOL := false;
    robot6axis_cams/cam_profile12/pFile AT 607 : DINT := 0;
    robot6axis_cams/cam_profile12/fault_reading AT 158 : BOOL := false;
    robot6axis_cams/cam_profile12/fault_openning AT 159 : BOOL := false;
    robot6axis_cams/cam_profile12/complete_path AT 3516 : STRING(254) := '';
    robot6axis_cams/cam_computation6/profileNr AT 523 : DINT := 0;
    robot6axis_cams/cam_computation6/MasterPositionIn AT 36 : REAL := 0.0;
    robot6axis_cams/cam_computation6/nbPoints0 AT 570 : INT := 0;
    robot6axis_cams/cam_computation6/MasterPoints0 AT 4671 : ARRAY[1..100] OF REAL := [100(0.0)];
    robot6axis_cams/cam_computation6/SlavePoints0 AT 4773 : ARRAY[1..100] OF REAL := [100(0.0)];
    robot6axis_cams/cam_computation6/pointer0 AT 571 : DINT := 0;
    robot6axis_cams/cam_computation6/nbPoints1 AT 572 : INT := 0;
    robot6axis_cams/cam_computation6/MasterPoints1 AT 4875 : ARRAY[1..100] OF REAL := [100(0.0)];
    robot6axis_cams/cam_computation6/SlavePoints1 AT 4977 : ARRAY[1..100] OF REAL := [100(0.0)];
    robot6axis_cams/cam_computation6/pointer1 AT 573 : DINT := 0;
    robot6axis_cams/cam_computation6/nbPoints2 AT 527 : INT := 0;
    robot6axis_cams/cam_computation6/MasterPoints2 AT 471 : ARRAY[1..100] OF REAL := [100(0.0)];
    robot6axis_cams/cam_computation6/SlavePoints2 AT 369 : ARRAY[1..100] OF REAL := [100(0.0)];
    robot6axis_cams/cam_computation6/pointer2 AT 526 : DINT := 0;
    robot6axis_cams/cam_computation6/nbPoints3 AT 525 : INT := 0;
    robot6axis_cams/cam_computation6/MasterPoints3 AT 267 : ARRAY[1..100] OF REAL := [100(0.0)];
    robot6axis_cams/cam_computation6/SlavePoints3 AT 165 : ARRAY[1..100] OF REAL := [100(0.0)];
    robot6axis_cams/cam_computation6/pointer3 AT 524 : DINT := 0;
    robot6axis_cams/cam_computation6/slavePosition AT 163 : REAL := 0.0;
    robot6axis_cams/cam_computation6/masterPosition AT 164 : REAL := 0.0;
    robot6axis_cams/cam_computation6/i AT 608 : INT := 0;
    robot6axis_cams/cam_computation6/modulo AT 6173 : REAL := 0.0;
    robot6axis_cams/cam_computation6/divider AT 609 : INT := 0;
    robot6axis_cams/cam_computation6/faultProfileNr AT 160 : BOOL := false;
    robot6axis_cams/cam_computation6/faultMasterPositionOOB AT 161 : BOOL := false;
    robot6axis_cams/cam_computation6/faultLinComputation AT 162 : BOOL := false;
    robot6axis_cams/cam_computation6/nbPoints AT 610 : INT := 0;
    robot6axis_cams/cam_computation6/MasterPoints AT 6174 : ARRAY[1..100] OF REAL := [100(0.0)];
    robot6axis_cams/cam_computation6/SlavePoints AT 6276 : ARRAY[1..100] OF REAL := [100(0.0)];
    robot6axis_cams/cam_computation6/found AT 163 : BOOL := false;
    robot6axis_cams/cam_computation6/index AT 611 : INT := 0;
    robot6axis_cams/cam_computation6/linDenom AT 6378 : REAL := 0.0;
    robot6axis_cams/cam_computation6/linNum AT 6379 : REAL := 0.0;
    robot6axis_cams/cam_computation6/linA AT 6380 : REAL := 0.0;
    robot6axis_cams/cam_computation6/linB AT 6381 : REAL := 0.0;
    robot6axis_cams/cam_computation6/FACTOR AT 6382 : REAL := 1.0;
    robot6axis/armOrigin AT 17 : ARRAY[1..3] OF REAL := [800.0, 400.0, 0.0];
    robot6axis/structRotVectorFOOT AT 153 : ARRAY[1..3] OF REAL := [0.0, 1.0, 0.0];
    robot6axis/structRotDegFOOT AT 152 : REAL := -90.01;
    robot6axis/ownRotDegFOOT AT 151 : REAL := 90.0;
    robot6axis/structRotVectorFOOT2 AT 146 : ARRAY[1..3] OF REAL := [2(0.0), 1.0];
    robot6axis/structRotDegFOOT2 AT 145 : REAL := 90.0;
    robot6axis/structRotVectorArm2 AT 140 : ARRAY[1..3] OF REAL := [2(0.0), 1.0];
    robot6axis/structRotDegArm2 AT 139 : REAL := -90.0;
    robot6axis/driveRotVector1 AT 134 : ARRAY[1..3] OF REAL := [1.0, 2(0.0)];
    robot6axis/driveRotVector2 AT 129 : ARRAY[1..3] OF REAL := [0.0, 1.0, 0.0];
    robot6axis/driveRotVector3 AT 124 : ARRAY[1..3] OF REAL := [0.0, 1.0, 0.0];
    robot6axis/driveRotVector4 AT 119 : ARRAY[1..3] OF REAL := [1.0, 2(0.0)];
    robot6axis/driveRotVector5 AT 114 : ARRAY[1..3] OF REAL := [0.0, 1.0, 0.0];
    robot6axis/driveRotVector6 AT 109 : ARRAY[1..3] OF REAL := [1.0, 2(0.0)];
    robot6axis/structRotVector1RowA AT 104 : ARRAY[1..3] OF REAL := [0.0, 1.0, 0.0];
    robot6axis/structRotDeg1RowA AT 103 : REAL := -90.0;
    robot6axis/structRotVector1RowB AT 98 : ARRAY[1..3] OF REAL := [0.0, 1.0, 0.0];
    robot6axis/structRotDeg1RowB AT 97 : REAL := 90.0;
    robot6axis/structRotVectorMultiRowsA AT 92 : ARRAY[1..3] OF REAL := [0.0, 1.0, 0.0];
    robot6axis/structRotDegMultiRowsA AT 91 : REAL := 90.0;
    robot6axis/structRotVectorMultiRowsB AT 86 : ARRAY[1..3] OF REAL := [0.0, 1.0, 0.0];
    robot6axis/structRotDegMultiRowsB AT 85 : REAL := -90.0;
    robot6axis/HomeCmd AT 77 : BOOL := false;
    robot6axis/MoveVelCmd AT 76 : BOOL := false;
    robot6axis/MoveAbsCmd AT 75 : BOOL := false;
    robot6axis/MoveVel1ManualCmd AT 74 : BOOL := false;
    robot6axis/MoveVel2ManualCmd AT 73 : BOOL := false;
    robot6axis/MoveAbs1ManualCmd AT 72 : BOOL := false;
    robot6axis/MoveAbs2ManualCmd AT 71 : BOOL := false;
    robot6axis/StopCmd AT 14 : BOOL := false;
    robot6axis/MovePosition AT 84 : REAL := 0.0;
    robot6axis/MoveSpeed AT 83 : REAL := 100.0;
    robot6axis/MoveAcceleration AT 82 : REAL := 100.0;
    robot6axis/MoveDeceleration AT 81 : REAL := 100.0;
    robot6axis/offsetAxToMa AT 80 : REAL := 0.0;
    robot6axis/HomeCmd2 AT 70 : BOOL := false;
    robot6axis/MoveVelCmd2 AT 69 : BOOL := false;
    robot6axis/MoveAbsCmd2 AT 68 : BOOL := false;
    robot6axis/MoveVel1ManualCmd2 AT 67 : BOOL := false;
    robot6axis/MoveVel2ManualCmd2 AT 66 : BOOL := false;
    robot6axis/MoveAbs1ManualCmd2 AT 65 : BOOL := false;
    robot6axis/MoveAbs2ManualCmd2 AT 64 : BOOL := false;
    robot6axis/StopCmd2 AT 14 : BOOL := false;
    robot6axis/MovePosition2 AT 79 : REAL := 0.0;
    robot6axis/MoveSpeed2 AT 78 : REAL := 100.0;
    robot6axis/MoveAcceleration2 AT 77 : REAL := 100.0;
    robot6axis/MoveDeceleration2 AT 76 : REAL := 100.0;
    robot6axis/offsetAxToMa2 AT 75 : REAL := 0.0;
    robot6axis/HomeCmd3 AT 63 : BOOL := false;
    robot6axis/MoveVelCmd3 AT 62 : BOOL := false;
    robot6axis/MoveAbsCmd3 AT 61 : BOOL := false;
    robot6axis/MoveVel1ManualCmd3 AT 60 : BOOL := false;
    robot6axis/MoveVel2ManualCmd3 AT 59 : BOOL := false;
    robot6axis/MoveAbs1ManualCmd3 AT 58 : BOOL := false;
    robot6axis/MoveAbs2ManualCmd3 AT 57 : BOOL := false;
    robot6axis/StopCmd3 AT 14 : BOOL := false;
    robot6axis/MovePosition3 AT 74 : REAL := 0.0;
    robot6axis/MoveSpeed3 AT 73 : REAL := 100.0;
    robot6axis/MoveAcceleration3 AT 72 : REAL := 100.0;
    robot6axis/MoveDeceleration3 AT 71 : REAL := 100.0;
    robot6axis/offsetAxToMa3 AT 70 : REAL := 0.0;
    robot6axis/HomeCmd4 AT 56 : BOOL := false;
    robot6axis/MoveVelCmd4 AT 55 : BOOL := false;
    robot6axis/MoveAbsCmd4 AT 54 : BOOL := false;
    robot6axis/MoveVel1ManualCmd4 AT 53 : BOOL := false;
    robot6axis/MoveVel2ManualCmd4 AT 52 : BOOL := false;
    robot6axis/MoveAbs1ManualCmd4 AT 51 : BOOL := false;
    robot6axis/MoveAbs2ManualCmd4 AT 50 : BOOL := false;
    robot6axis/StopCmd4 AT 14 : BOOL := false;
    robot6axis/MovePosition4 AT 69 : REAL := 0.0;
    robot6axis/MoveSpeed4 AT 68 : REAL := 100.0;
    robot6axis/MoveAcceleration4 AT 67 : REAL := 100.0;
    robot6axis/MoveDeceleration4 AT 66 : REAL := 100.0;
    robot6axis/offsetAxToMa4 AT 65 : REAL := 0.0;
    robot6axis/HomeCmd5 AT 49 : BOOL := false;
    robot6axis/MoveVelCmd5 AT 48 : BOOL := false;
    robot6axis/MoveAbsCmd5 AT 47 : BOOL := false;
    robot6axis/MoveVel1ManualCmd5 AT 46 : BOOL := false;
    robot6axis/MoveVel2ManualCmd5 AT 45 : BOOL := false;
    robot6axis/MoveAbs1ManualCmd5 AT 44 : BOOL := false;
    robot6axis/MoveAbs2ManualCmd5 AT 43 : BOOL := false;
    robot6axis/StopCmd5 AT 14 : BOOL := false;
    robot6axis/MovePosition5 AT 64 : REAL := 0.0;
    robot6axis/MoveSpeed5 AT 63 : REAL := 100.0;
    robot6axis/MoveAcceleration5 AT 62 : REAL := 100.0;
    robot6axis/MoveDeceleration5 AT 61 : REAL := 100.0;
    robot6axis/offsetAxToMa5 AT 60 : REAL := 0.0;
    robot6axis/HomeCmd6 AT 42 : BOOL := false;
    robot6axis/MoveVelCmd6 AT 41 : BOOL := false;
    robot6axis/MoveAbsCmd6 AT 40 : BOOL := false;
    robot6axis/MoveVel1ManualCmd6 AT 39 : BOOL := false;
    robot6axis/MoveVel2ManualCmd6 AT 38 : BOOL := false;
    robot6axis/MoveAbs1ManualCmd6 AT 37 : BOOL := false;
    robot6axis/MoveAbs2ManualCmd6 AT 36 : BOOL := false;
    robot6axis/StopCmd6 AT 14 : BOOL := false;
    robot6axis/MovePosition6 AT 59 : REAL := 0.0;
    robot6axis/MoveSpeed6 AT 58 : REAL := 100.0;
    robot6axis/MoveAcceleration6 AT 57 : REAL := 100.0;
    robot6axis/MoveDeceleration6 AT 56 : REAL := 100.0;
    robot6axis/offsetAxToMa6 AT 55 : REAL := 0.0;
    robot6axis/PLC_StatusReady AT 35 : BOOL := true;
    robot6axis/PLC_StatusMoved AT 34 : BOOL := false;
    robot6axis/PLC_StatusStand AT 33 : BOOL := false;
    robot6axis/PLC_ActualPositionAx AT 158 : REAL := 0.0;
    robot6axis/PLC_ActualPositionMa AT 54 : REAL := 0.0;
    robot6axis/PLC_ActualVelocity AT 53 : REAL := 0.0;
    robot6axis/PLC_StatusReady2 AT 32 : BOOL := true;
    robot6axis/PLC_StatusMoved2 AT 31 : BOOL := false;
    robot6axis/PLC_StatusStand2 AT 30 : BOOL := false;
    robot6axis/PLC_ActualPositionAx2 AT 159 : REAL := 0.0;
    robot6axis/PLC_ActualPositionMa2 AT 52 : REAL := 0.0;
    robot6axis/PLC_ActualVelocity2 AT 51 : REAL := 0.0;
    robot6axis/PLC_StatusReady3 AT 29 : BOOL := true;
    robot6axis/PLC_StatusMoved3 AT 28 : BOOL := false;
    robot6axis/PLC_StatusStand3 AT 27 : BOOL := false;
    robot6axis/PLC_ActualPositionAx3 AT 160 : REAL := 0.0;
    robot6axis/PLC_ActualPositionMa3 AT 50 : REAL := 0.0;
    robot6axis/PLC_ActualVelocity3 AT 49 : REAL := 0.0;
    robot6axis/PLC_StatusReady4 AT 26 : BOOL := true;
    robot6axis/PLC_StatusMoved4 AT 25 : BOOL := false;
    robot6axis/PLC_StatusStand4 AT 24 : BOOL := false;
    robot6axis/PLC_ActualPositionAx4 AT 161 : REAL := 0.0;
    robot6axis/PLC_ActualPositionMa4 AT 48 : REAL := 0.0;
    robot6axis/PLC_ActualVelocity4 AT 47 : REAL := 0.0;
    robot6axis/PLC_StatusReady5 AT 23 : BOOL := true;
    robot6axis/PLC_StatusMoved5 AT 22 : BOOL := false;
    robot6axis/PLC_StatusStand5 AT 21 : BOOL := false;
    robot6axis/PLC_ActualPositionAx5 AT 162 : REAL := 0.0;
    robot6axis/PLC_ActualPositionMa5 AT 46 : REAL := 0.0;
    robot6axis/PLC_ActualVelocity5 AT 45 : REAL := 0.0;
    robot6axis/PLC_StatusReady6 AT 20 : BOOL := true;
    robot6axis/PLC_StatusMoved6 AT 19 : BOOL := false;
    robot6axis/PLC_StatusStand6 AT 18 : BOOL := false;
    robot6axis/PLC_ActualPositionAx6 AT 163 : REAL := 0.0;
    robot6axis/PLC_ActualPositionMa6 AT 44 : REAL := 0.0;
    robot6axis/PLC_ActualVelocity6 AT 43 : REAL := 0.0;
    robot6axis/gripSyringes AT 13 : BOOL := false;
    robot6axis/ActualVelocity1 AT 42 : REAL := 0.0;
    robot6axis/ActualVelocity2 AT 41 : REAL := 0.0;
    robot6axis/ActualVelocity3 AT 40 : REAL := 0.0;
    robot6axis/ActualVelocity4 AT 39 : REAL := 0.0;
    robot6axis/ActualVelocity5 AT 38 : REAL := 0.0;
    robot6axis/ActualVelocity6 AT 37 : REAL := 0.0;
    robot6axis/armExtrem AT 27 : ARRAY[1..3] OF REAL := [3(0.0)];
    robot6axis/velX AT 32 : REAL := 0.0;
    robot6axis/velY AT 33 : REAL := 0.0;
    robot6axis/velZ AT 34 : REAL := 0.0;
    robot6axis/armInStop AT 17 : BOOL := false;
    robot6axis/servo_1/status AT 631 : INT := 0;
    robot6axis/servo_1/errorFlag AT 630 : INT := 0;
    robot6axis/servo_1/ActualPositionAx1 AT 6518 : REAL := 0.0;
    robot6axis/servo_1/MoveVelDone1 AT 213 : BOOL := false;
    robot6axis/servo_1/ActualVelocity1 AT 6517 : REAL := 0.0;
    robot6axis/servo_1/MoveAbsDone1 AT 212 : BOOL := false;
    robot6axis/servo_1/HomeCmd AT 77 : BOOL := false;
    robot6axis/servo_1/MoveVelCmd AT 76 : BOOL := false;
    robot6axis/servo_1/MoveAbsCmd AT 75 : BOOL := false;
    robot6axis/servo_1/MoveVel1ManualCmd AT 74 : BOOL := false;
    robot6axis/servo_1/MoveVel2ManualCmd AT 73 : BOOL := false;
    robot6axis/servo_1/MoveAbs1ManualCmd AT 72 : BOOL := false;
    robot6axis/servo_1/MoveAbs2ManualCmd AT 71 : BOOL := false;
    robot6axis/servo_1/StopCmd AT 14 : BOOL := false;
    robot6axis/servo_1/MovePosition AT 84 : REAL := 0.0;
    robot6axis/servo_1/MoveSpeed AT 83 : REAL := 100.0;
    robot6axis/servo_1/MoveAcceleration AT 82 : REAL := 100.0;
    robot6axis/servo_1/MoveDeceleration AT 81 : REAL := 100.0;
    robot6axis/servo_1/offsetAxToMa AT 80 : REAL := 0.0;
    robot6axis/servo_1/PLC_StatusReady AT 35 : BOOL := true;
    robot6axis/servo_1/PLC_StatusMoved AT 34 : BOOL := false;
    robot6axis/servo_1/PLC_StatusStand AT 33 : BOOL := false;
    robot6axis/servo_1/PLC_ActualPositionAx AT 158 : REAL := 0.0;
    robot6axis/servo_1/PLC_ActualPositionMa AT 54 : REAL := 0.0;
    robot6axis/servo_1/PLC_ActualVelocity AT 53 : REAL := 0.0;
    robot6axis/servo_1/physicalPosInit AT 6516 : REAL := 0.0;
    robot6axis/servo_1/MAX_SPEED AT 6515 : REAL(0.0..3.4e+038) := 30.0;
    robot6axis/servo_1/MAX_ACCEL AT 6514 : REAL(0.0..3.4e+038) := 1500.0;
    robot6axis/servo_1/MAX_DECEL AT 6513 : REAL(0.0..3.4e+038) := 1500.0;
    robot6axis/servo_1/MODULO_LENGTH AT 6512 : REAL := 0.0;
    robot6axis/servo_1/StatusReady AT 211 : BOOL := true;
    robot6axis/servo_1/StatusMoved AT 210 : BOOL := false;
    robot6axis/servo_1/StatusStand AT 209 : BOOL := false;
    robot6axis/servo_1/ActualPositionAx AT 6519 : REAL := 0.0;
    robot6axis/servo_1/ActualPositionMa AT 6511 : REAL := 0.0;
    robot6axis/servo_1/ActualVelocity AT 42 : REAL := 0.0;
    robot6axis/servo_1/MaximumVelocity AT 6510 : REAL := 0.0;
    robot6axis/servo_1/StatusPosIncrease AT 208 : BOOL := false;
    robot6axis/servo_1/StatusPosDecrease AT 207 : BOOL := false;
    robot6axis/servo_1/displayJauge AT 6509 : REAL := 0.0;
    robot6axis/servo_1/servo_mode/PLC_StatusReady AT 35 : BOOL := true;
    robot6axis/servo_1/servo_mode/PLC_StatusMoved AT 34 : BOOL := false;
    robot6axis/servo_1/servo_mode/PLC_StatusStand AT 33 : BOOL := false;
    robot6axis/servo_1/servo_mode/PLC_ActualPositionAx AT 158 : REAL := 0.0;
    robot6axis/servo_1/servo_mode/PLC_ActualPositionMa AT 54 : REAL := 0.0;
    robot6axis/servo_1/servo_mode/PLC_ActualVelocity AT 53 : REAL := 0.0;
    robot6axis/servo_1/servo_mode/StatusReady AT 214 : BOOL := true;
    robot6axis/servo_1/servo_mode/StatusMoved AT 215 : BOOL := false;
    robot6axis/servo_1/servo_mode/StatusStand AT 216 : BOOL := false;
    robot6axis/servo_1/servo_mode/ActualPositionMa AT 6608 : REAL := 0.0;
    robot6axis/servo_1/servo_mode/ActualVelocity AT 6609 : REAL := 0.0;
    robot6axis/servo_1/servo_mode/MaximumVelocity AT 6610 : REAL := 0.0;
    robot6axis/servo_1/servo_mode/physicalPosInit AT 6516 : REAL := 0.0;
    robot6axis/servo_1/servo_mode/ActualPositionAx AT 6518 : REAL := 0.0;
    robot6axis/servo_1/servo_mode/StatusReady_o AT 211 : BOOL := true;
    robot6axis/servo_1/servo_mode/StatusMoved_o AT 210 : BOOL := false;
    robot6axis/servo_1/servo_mode/StatusStand_o AT 209 : BOOL := false;
    robot6axis/servo_1/servo_mode/ActualPositionAx_o AT 6519 : REAL := 0.0;
    robot6axis/servo_1/servo_mode/ActualPositionMa_o AT 6511 : REAL := 0.0;
    robot6axis/servo_1/servo_mode/ActualVelocity_o AT 42 : REAL := 0.0;
    robot6axis/servo_1/servo_mode/MaximumVelocity_o AT 6510 : REAL := 0.0;
    robot6axis/servo_1/servo_mode/StatusPosIncrease_o AT 208 : BOOL := false;
    robot6axis/servo_1/servo_mode/StatusPosDecrease_o AT 207 : BOOL := false;
    robot6axis/servo_1/servo_mode/displayJauge_o AT 6509 : REAL := 0.0;
    robot6axis/servo_1/servo_mode/PLCMode AT 221 : BOOL := false;
    robot6axis/servo_1/servo_mode/PLCMode1 AT 222 : BOOL := false;
    robot6axis/servo_1/servo_mode/initDone AT 223 : BOOL := false;
    robot6axis/servo_1/servo_mode/displayPosMin AT 6613 : REAL := 0.0;
    robot6axis/servo_1/servo_mode/displayPosMax AT 6614 : REAL := 0.0;
    robot6axis/servo_1/servo_mode/PLC_ActualPositionAx1 AT 6615 : REAL := 0.0;
    robot6axis/servo_1/servo_mode/PLC_ActualVelocity1 AT 6616 : REAL := 0.0;
    robot6axis/servo_1/servo_mode/ActualPositionAx1 AT 6617 : REAL := 0.0;
    robot6axis/servo_1/servo_mode/ActualVelocity1 AT 6618 : REAL := 0.0;
    robot6axis/servo_1/servo_mode/offsetAxToMa AT 6619 : REAL := 0.0;
    robot6axis/servo_1/servo_mode/offsetAxToMa1 AT 6620 : REAL := 0.0;
    robot6axis/servo_1/servo_mode/ActualPositionMa_o1 AT 6621 : REAL := 0.0;
    robot6axis/servo_1/servo_control/HomeCmd AT 77 : BOOL := false;
    robot6axis/servo_1/servo_control/MoveVelCmd AT 76 : BOOL := false;
    robot6axis/servo_1/servo_control/MoveAbsCmd AT 75 : BOOL := false;
    robot6axis/servo_1/servo_control/MoveVel1ManualCmd AT 74 : BOOL := false;
    robot6axis/servo_1/servo_control/MoveVel2ManualCmd AT 73 : BOOL := false;
    robot6axis/servo_1/servo_control/MoveAbs1ManualCmd AT 72 : BOOL := false;
    robot6axis/servo_1/servo_control/MoveAbs2ManualCmd AT 71 : BOOL := false;
    robot6axis/servo_1/servo_control/StopCmd AT 14 : BOOL := false;
    robot6axis/servo_1/servo_control/MovePosition AT 84 : REAL := 0.0;
    robot6axis/servo_1/servo_control/MoveSpeed AT 83 : REAL := 100.0;
    robot6axis/servo_1/servo_control/MoveAcceleration AT 82 : REAL := 100.0;
    robot6axis/servo_1/servo_control/MoveDeceleration AT 81 : REAL := 100.0;
    robot6axis/servo_1/servo_control/offsetAxToMa AT 80 : REAL := 0.0;
    robot6axis/servo_1/servo_control/physicalPosInit AT 6516 : REAL := 0.0;
    robot6axis/servo_1/servo_control/MAX_SPEED AT 6515 : REAL(0.0..3.4e+038) := 30.0;
    robot6axis/servo_1/servo_control/status AT 631 : INT := 0;
    robot6axis/servo_1/servo_control/errorFlag AT 630 : INT := 0;
    robot6axis/servo_1/servo_control/IOActualPositionAx AT 6518 : REAL := 0.0;
    robot6axis/servo_1/servo_control/IOVelDone AT 213 : BOOL := false;
    robot6axis/servo_1/servo_control/IOAbsDone AT 212 : BOOL := false;
    robot6axis/servo_1/servo_control/IOActualVelocity AT 6517 : REAL := 0.0;
    robot6axis/servo_1/servo_control/OperationMode AT 633 : INT := 0;
    robot6axis/servo_1/servo_control/StatusReady AT 214 : BOOL := true;
    robot6axis/servo_1/servo_control/StatusMove AT 215 : BOOL := false;
    robot6axis/servo_1/servo_control/StatusStand AT 216 : BOOL := false;
    robot6axis/servo_1/servo_control/ActualPositionMa AT 6608 : REAL := 0.0;
    robot6axis/servo_1/servo_control/ActualVelocity AT 6609 : REAL := 0.0;
    robot6axis/servo_1/servo_control/MaximumVelocity AT 6610 : REAL := 0.0;
    robot6axis/servo_1/servo_control/VelEnabled AT 217 : BOOL := false;
    robot6axis/servo_1/servo_control/VelCmd AT 218 : BOOL := false;
    robot6axis/servo_1/servo_control/PosEnabled AT 219 : BOOL := false;
    robot6axis/servo_1/servo_control/PosCmd AT 220 : BOOL := false;
    robot6axis/servo_1/servo_control/Position AT 6612 : REAL := 0.0;
    robot6axis/servo_1/servo_control/Speed AT 6611 : REAL := 0.0;
    robot6axis/servo_1/servo_control/ManualMode AT 634 : INT := 0;
    robot6axis/servo_1/servo_control/initDone AT 224 : BOOL := false;
    robot6axis/servo_1/servo_control/ActualPositionMa1 AT 6622 : REAL := 0.0;
    robot6axis/servo_1/servo_control/offsetAxToMa1 AT 6623 : REAL := 0.0;
    robot6axis/servo_1/servo_control/HOME_POSITION AT 6624 : REAL := 100.0;
    robot6axis/servo_1/servo_control/MANUAL_POSITION1 AT 6625 : REAL := 0.0;
    robot6axis/servo_1/servo_control/MANUAL_POSITION2 AT 6626 : REAL := 150.0;
    robot6axis/servo_1/servo_control/MANUAL_SPEED1 AT 6627 : REAL := -100.0;
    robot6axis/servo_1/servo_control/MANUAL_SPEED2 AT 6628 : REAL := 100.0;
    robot6axis/servo_1/servo_control/MANUAL_SPEED AT 6629 : REAL := 100.0;
    robot6axis/servo_1/servo_velocity/MoveVelEnable AT 217 : BOOL := false;
    robot6axis/servo_1/servo_velocity/MoveVelStart AT 218 : BOOL := false;
    robot6axis/servo_1/servo_velocity/MoveSpeed AT 6611 : REAL := 0.0;
    robot6axis/servo_1/servo_velocity/MoveAcceleration AT 82 : REAL := 100.0;
    robot6axis/servo_1/servo_velocity/MoveDeceleration AT 81 : REAL := 100.0;
    robot6axis/servo_1/servo_velocity/MAX_SPEED AT 6515 : REAL(0.0..3.4e+038) := 30.0;
    robot6axis/servo_1/servo_velocity/MAX_ACCEL AT 6514 : REAL(0.0..3.4e+038) := 1500.0;
    robot6axis/servo_1/servo_velocity/MAX_DECEL AT 6513 : REAL(0.0..3.4e+038) := 1500.0;
    robot6axis/servo_1/servo_velocity/MODULO_LENGTH AT 6512 : REAL := 0.0;
    robot6axis/servo_1/servo_velocity/status AT 631 : INT := 0;
    robot6axis/servo_1/servo_velocity/errorFlag AT 630 : INT := 0;
    robot6axis/servo_1/servo_velocity/MoveVelDone AT 213 : BOOL := false;
    robot6axis/servo_1/servo_velocity/ActualPositionAx AT 6518 : REAL := 0.0;
    robot6axis/servo_1/servo_velocity/ActualVelocity AT 6517 : REAL := 0.0;
    robot6axis/servo_1/servo_velocity/firstStep AT 225 : BOOL := true;
    robot6axis/servo_1/servo_velocity/stepDone AT 226 : BOOL := false;
    robot6axis/servo_1/servo_velocity/currentTime AT 6630 : REAL := 0.0;
    robot6axis/servo_1/servo_velocity/MoveSpeed1 AT 6631 : REAL := 0.0;
    robot6axis/servo_1/servo_velocity/acceleration AT 6632 : REAL := 0.0;
    robot6axis/servo_1/servo_velocity/deceleration AT 6633 : REAL := 0.0;
    robot6axis/servo_1/servo_velocity/orderSpeed AT 6634 : REAL := 0.0;
    robot6axis/servo_1/servo_velocity/endChangeSpeed AT 6635 : REAL := 0.0;
    robot6axis/servo_1/servo_velocity/accelDecelChangeSpeed AT 6636 : REAL := 0.0;
    robot6axis/servo_1/servo_velocity/ActualVelocity1 AT 6637 : REAL := 0.0;
    robot6axis/servo_1/servo_velocity/speedChanged AT 227 : BOOL := false;
    robot6axis/servo_1/servo_position/MoveAbsEnable AT 219 : BOOL := false;
    robot6axis/servo_1/servo_position/MoveAbsStart AT 220 : BOOL := false;
    robot6axis/servo_1/servo_position/MovePosition AT 6612 : REAL := 0.0;
    robot6axis/servo_1/servo_position/MoveSpeed AT 6611 : REAL := 0.0;
    robot6axis/servo_1/servo_position/MoveAcceleration AT 82 : REAL := 100.0;
    robot6axis/servo_1/servo_position/MoveDeceleration AT 81 : REAL := 100.0;
    robot6axis/servo_1/servo_position/MAX_SPEED AT 6515 : REAL(0.0..3.4e+038) := 30.0;
    robot6axis/servo_1/servo_position/MAX_ACCEL AT 6514 : REAL(0.0..3.4e+038) := 1500.0;
    robot6axis/servo_1/servo_position/MAX_DECEL AT 6513 : REAL(0.0..3.4e+038) := 1500.0;
    robot6axis/servo_1/servo_position/MODULO_LENGTH AT 6512 : REAL := 0.0;
    robot6axis/servo_1/servo_position/status AT 631 : INT := 0;
    robot6axis/servo_1/servo_position/errorFlag AT 630 : INT := 0;
    robot6axis/servo_1/servo_position/MoveAbsDone AT 212 : BOOL := false;
    robot6axis/servo_1/servo_position/ActualPositionAx AT 6518 : REAL := 0.0;
    robot6axis/servo_1/servo_position/ActualVelocity AT 6517 : REAL := 0.0;
    robot6axis/servo_1/servo_position/firstStep AT 228 : BOOL := true;
    robot6axis/servo_1/servo_position/stepDone AT 229 : BOOL := false;
    robot6axis/servo_1/servo_position/timeToStop AT 6638 : REAL := 0.0;
    robot6axis/servo_1/servo_position/distanceToStop AT 6639 : REAL := 0.0;
    robot6axis/servo_1/servo_position/distance AT 6640 : REAL := 0.0;
    robot6axis/servo_1/servo_position/currentTime AT 6641 : REAL := 0.0;
    robot6axis/servo_1/servo_position/currentSpeed1 AT 6642 : REAL := 0.0;
    robot6axis/servo_1/servo_position/targetPosition AT 6643 : REAL := 0.0;
    robot6axis/servo_1/servo_position/ActualPositionAx1 AT 6644 : REAL := 0.0;
    robot6axis/servo_1/servo_position/acceleration AT 6645 : REAL := 0.0;
    robot6axis/servo_1/servo_position/deceleration AT 6646 : REAL := 0.0;
    robot6axis/servo_1/servo_position/orderSpeed AT 6647 : REAL := 0.0;
    robot6axis/servo_1/servo_position/moveDirection AT 6648 : REAL := 0.0;
    robot6axis/servo_1/servo_position/moveDirection1 AT 6649 : REAL := 0.0;
    robot6axis/servo_1/servo_position/endChangeSpeed AT 6650 : REAL := 0.0;
    robot6axis/servo_1/servo_position/ActualVelocity1 AT 6651 : REAL := 0.0;
    robot6axis/FOOT/armOrigin AT 17 : ARRAY[1..3] OF REAL := [800.0, 400.0, 0.0];
    robot6axis/FOOT/overallArmQuatInput AT 6503 : ARRAY[1..4] OF REAL := [1.0, 3(0.0)];
    robot6axis/FOOT/structRotVector AT 153 : ARRAY[1..3] OF REAL := [0.0, 1.0, 0.0];
    robot6axis/FOOT/structRotDeg AT 152 : REAL := -90.01;
    robot6axis/FOOT/driveRotVector AT 134 : ARRAY[1..3] OF REAL := [1.0, 2(0.0)];
    robot6axis/FOOT/driveRotDeg AT 6519 : REAL := 0.0;
    robot6axis/FOOT/ownRotDeg AT 151 : REAL := 90.0;
    robot6axis/FOOT/driveResizeLength AT 6502 : REAL := 0.0;
    robot6axis/FOOT/functionActive AT 206 : BOOL := false;
    robot6axis/FOOT/armExtrem AT 6520 : ARRAY[1..3] OF REAL := [3(0.0)];
    robot6axis/FOOT/overallArmRotOutput AT 6525 : ARRAY[1..4] OF REAL := [4(0.0)];
    robot6axis/FOOT/productId AT 629 : DINT := -1;
    robot6axis/FOOT/status_act_prod AT 635 : DINT := 0;
    robot6axis/FOOT/m11 AT 6652 : REAL := 56.5871;
    robot6axis/FOOT/m12 AT 6653 : REAL := 0.0;
    robot6axis/FOOT/m13 AT 6654 : REAL := 0.0;
    robot6axis/FOOT/m14 AT 6655 : REAL := 25.4642;
    robot6axis/FOOT/m21 AT 6656 : REAL := 0.0;
    robot6axis/FOOT/m22 AT 6657 : REAL := 35.0133;
    robot6axis/FOOT/m23 AT 6658 : REAL := 0.0;
    robot6axis/FOOT/m24 AT 6659 : REAL := 96.1981;
    robot6axis/FOOT/m31 AT 6660 : REAL := 0.0;
    robot6axis/FOOT/m32 AT 6661 : REAL := 0.0;
    robot6axis/FOOT/m33 AT 6662 : REAL := 14.1468;
    robot6axis/FOOT/m34 AT 6663 : REAL := 74.2706;
    robot6axis/FOOT/m41 AT 6664 : REAL := 0.0;
    robot6axis/FOOT/m42 AT 6665 : REAL := 0.0;
    robot6axis/FOOT/m43 AT 6666 : REAL := 0.0;
    robot6axis/FOOT/m44 AT 6667 : REAL := 1.0;
    robot6axis/FOOT/armLengthCalc AT 6668 : REAL := 0.0;
    robot6axis/FOOT/functionActiveLocale AT 230 : BOOL := false;
    robot6axis/FOOT/product_id AT 636 : DINT := -1;
    robot6axis/FOOT/arm_id AT 637 : DINT := -1;
    robot6axis/FOOT/timeToGripParam AT 6669 : REAL := 0.15;
    robot6axis/FOOT/armLength AT 6670 : REAL := 375.0;
    robot6axis/FOOT/armWidth AT 6671 : REAL := 60.0;
    robot6axis/FOOT/armHeight AT 6672 : REAL := 60.0;
    robot6axis/FOOT/armType AT 638 : INT := 0;
    robot6axis/FOOT2/armOrigin AT 6520 : ARRAY[1..3] OF REAL := [3(0.0)];
    robot6axis/FOOT2/overallArmQuatInput AT 6525 : ARRAY[1..4] OF REAL := [4(0.0)];
    robot6axis/FOOT2/structRotVector AT 146 : ARRAY[1..3] OF REAL := [2(0.0), 1.0];
    robot6axis/FOOT2/structRotDeg AT 145 : REAL := 90.0;
    robot6axis/FOOT2/driveRotVector AT 6497 : ARRAY[1..3] OF REAL := [2(0.0), 1.0];
    robot6axis/FOOT2/driveRotDeg AT 6496 : REAL := 0.0;
    robot6axis/FOOT2/ownRotDeg AT 6495 : REAL := 0.0;
    robot6axis/FOOT2/driveResizeLength AT 6494 : REAL := 0.0;
    robot6axis/FOOT2/functionActive AT 205 : BOOL := false;
    robot6axis/FOOT2/armExtrem AT 6531 : ARRAY[1..3] OF REAL := [3(0.0)];
    robot6axis/FOOT2/overallArmRotOutput AT 6536 : ARRAY[1..4] OF REAL := [4(0.0)];
    robot6axis/FOOT2/productId AT 628 : DINT := -1;
    robot6axis/FOOT2/status_act_prod AT 639 : DINT := 0;
    robot6axis/FOOT2/m11 AT 6673 : REAL := 1.0;
    robot6axis/FOOT2/m12 AT 6674 : REAL := 0.0;
    robot6axis/FOOT2/m13 AT 6675 : REAL := 0.0;
    robot6axis/FOOT2/m14 AT 6676 : REAL := 0.0;
    robot6axis/FOOT2/m21 AT 6677 : REAL := 0.0;
    robot6axis/FOOT2/m22 AT 6678 : REAL := 1.0;
    robot6axis/FOOT2/m23 AT 6679 : REAL := 0.0;
    robot6axis/FOOT2/m24 AT 6680 : REAL := 0.0;
    robot6axis/FOOT2/m31 AT 6681 : REAL := 0.0;
    robot6axis/FOOT2/m32 AT 6682 : REAL := 0.0;
    robot6axis/FOOT2/m33 AT 6683 : REAL := 1.0;
    robot6axis/FOOT2/m34 AT 6684 : REAL := 0.0;
    robot6axis/FOOT2/m41 AT 6685 : REAL := 0.0;
    robot6axis/FOOT2/m42 AT 6686 : REAL := 0.0;
    robot6axis/FOOT2/m43 AT 6687 : REAL := 0.0;
    robot6axis/FOOT2/m44 AT 6688 : REAL := 1.0;
    robot6axis/FOOT2/armLengthCalc AT 6689 : REAL := 0.0;
    robot6axis/FOOT2/functionActiveLocale AT 231 : BOOL := false;
    robot6axis/FOOT2/product_id AT 640 : DINT := -1;
    robot6axis/FOOT2/arm_id AT 641 : DINT := -1;
    robot6axis/FOOT2/timeToGripParam AT 6690 : REAL := 0.15;
    robot6axis/FOOT2/armLength AT 6691 : REAL := 20.0;
    robot6axis/FOOT2/armWidth AT 6692 : REAL := 60.0;
    robot6axis/FOOT2/armHeight AT 6693 : REAL := 60.0;
    robot6axis/FOOT2/armType AT 642 : INT := 0;
    robot6axis/servo_2/status AT 627 : INT := 0;
    robot6axis/servo_2/errorFlag AT 626 : INT := 0;
    robot6axis/servo_2/ActualPositionAx1 AT 6493 : REAL := 0.0;
    robot6axis/servo_2/MoveVelDone1 AT 204 : BOOL := false;
    robot6axis/servo_2/ActualVelocity1 AT 6492 : REAL := 0.0;
    robot6axis/servo_2/MoveAbsDone1 AT 203 : BOOL := false;
    robot6axis/servo_2/HomeCmd AT 70 : BOOL := false;
    robot6axis/servo_2/MoveVelCmd AT 69 : BOOL := false;
    robot6axis/servo_2/MoveAbsCmd AT 68 : BOOL := false;
    robot6axis/servo_2/MoveVel1ManualCmd AT 67 : BOOL := false;
    robot6axis/servo_2/MoveVel2ManualCmd AT 66 : BOOL := false;
    robot6axis/servo_2/MoveAbs1ManualCmd AT 65 : BOOL := false;
    robot6axis/servo_2/MoveAbs2ManualCmd AT 64 : BOOL := false;
    robot6axis/servo_2/StopCmd AT 14 : BOOL := false;
    robot6axis/servo_2/MovePosition AT 79 : REAL := 0.0;
    robot6axis/servo_2/MoveSpeed AT 78 : REAL := 100.0;
    robot6axis/servo_2/MoveAcceleration AT 77 : REAL := 100.0;
    robot6axis/servo_2/MoveDeceleration AT 76 : REAL := 100.0;
    robot6axis/servo_2/offsetAxToMa AT 75 : REAL := 0.0;
    robot6axis/servo_2/PLC_StatusReady AT 32 : BOOL := true;
    robot6axis/servo_2/PLC_StatusMoved AT 31 : BOOL := false;
    robot6axis/servo_2/PLC_StatusStand AT 30 : BOOL := false;
    robot6axis/servo_2/PLC_ActualPositionAx AT 159 : REAL := 0.0;
    robot6axis/servo_2/PLC_ActualPositionMa AT 52 : REAL := 0.0;
    robot6axis/servo_2/PLC_ActualVelocity AT 51 : REAL := 0.0;
    robot6axis/servo_2/physicalPosInit AT 6491 : REAL := 0.0;
    robot6axis/servo_2/MAX_SPEED AT 6490 : REAL(0.0..3.4e+038) := 30.0;
    robot6axis/servo_2/MAX_ACCEL AT 6489 : REAL(0.0..3.4e+038) := 1500.0;
    robot6axis/servo_2/MAX_DECEL AT 6488 : REAL(0.0..3.4e+038) := 1500.0;
    robot6axis/servo_2/MODULO_LENGTH AT 6487 : REAL := 0.0;
    robot6axis/servo_2/StatusReady AT 202 : BOOL := true;
    robot6axis/servo_2/StatusMoved AT 201 : BOOL := false;
    robot6axis/servo_2/StatusStand AT 200 : BOOL := false;
    robot6axis/servo_2/ActualPositionAx AT 6542 : REAL := 0.0;
    robot6axis/servo_2/ActualPositionMa AT 6486 : REAL := 0.0;
    robot6axis/servo_2/ActualVelocity AT 41 : REAL := 0.0;
    robot6axis/servo_2/MaximumVelocity AT 6485 : REAL := 0.0;
    robot6axis/servo_2/StatusPosIncrease AT 199 : BOOL := false;
    robot6axis/servo_2/StatusPosDecrease AT 198 : BOOL := false;
    robot6axis/servo_2/displayJauge AT 6484 : REAL := 0.0;
    robot6axis/servo_2/servo_mode/PLC_StatusReady AT 32 : BOOL := true;
    robot6axis/servo_2/servo_mode/PLC_StatusMoved AT 31 : BOOL := false;
    robot6axis/servo_2/servo_mode/PLC_StatusStand AT 30 : BOOL := false;
    robot6axis/servo_2/servo_mode/PLC_ActualPositionAx AT 159 : REAL := 0.0;
    robot6axis/servo_2/servo_mode/PLC_ActualPositionMa AT 52 : REAL := 0.0;
    robot6axis/servo_2/servo_mode/PLC_ActualVelocity AT 51 : REAL := 0.0;
    robot6axis/servo_2/servo_mode/StatusReady AT 232 : BOOL := true;
    robot6axis/servo_2/servo_mode/StatusMoved AT 233 : BOOL := false;
    robot6axis/servo_2/servo_mode/StatusStand AT 234 : BOOL := false;
    robot6axis/servo_2/servo_mode/ActualPositionMa AT 6694 : REAL := 0.0;
    robot6axis/servo_2/servo_mode/ActualVelocity AT 6695 : REAL := 0.0;
    robot6axis/servo_2/servo_mode/MaximumVelocity AT 6696 : REAL := 0.0;
    robot6axis/servo_2/servo_mode/physicalPosInit AT 6491 : REAL := 0.0;
    robot6axis/servo_2/servo_mode/ActualPositionAx AT 6493 : REAL := 0.0;
    robot6axis/servo_2/servo_mode/StatusReady_o AT 202 : BOOL := true;
    robot6axis/servo_2/servo_mode/StatusMoved_o AT 201 : BOOL := false;
    robot6axis/servo_2/servo_mode/StatusStand_o AT 200 : BOOL := false;
    robot6axis/servo_2/servo_mode/ActualPositionAx_o AT 6542 : REAL := 0.0;
    robot6axis/servo_2/servo_mode/ActualPositionMa_o AT 6486 : REAL := 0.0;
    robot6axis/servo_2/servo_mode/ActualVelocity_o AT 41 : REAL := 0.0;
    robot6axis/servo_2/servo_mode/MaximumVelocity_o AT 6485 : REAL := 0.0;
    robot6axis/servo_2/servo_mode/StatusPosIncrease_o AT 199 : BOOL := false;
    robot6axis/servo_2/servo_mode/StatusPosDecrease_o AT 198 : BOOL := false;
    robot6axis/servo_2/servo_mode/displayJauge_o AT 6484 : REAL := 0.0;
    robot6axis/servo_2/servo_mode/PLCMode AT 239 : BOOL := false;
    robot6axis/servo_2/servo_mode/PLCMode1 AT 240 : BOOL := false;
    robot6axis/servo_2/servo_mode/initDone AT 241 : BOOL := false;
    robot6axis/servo_2/servo_mode/displayPosMin AT 6699 : REAL := 0.0;
    robot6axis/servo_2/servo_mode/displayPosMax AT 6700 : REAL := 0.0;
    robot6axis/servo_2/servo_mode/PLC_ActualPositionAx1 AT 6701 : REAL := 0.0;
    robot6axis/servo_2/servo_mode/PLC_ActualVelocity1 AT 6702 : REAL := 0.0;
    robot6axis/servo_2/servo_mode/ActualPositionAx1 AT 6703 : REAL := 0.0;
    robot6axis/servo_2/servo_mode/ActualVelocity1 AT 6704 : REAL := 0.0;
    robot6axis/servo_2/servo_mode/offsetAxToMa AT 6705 : REAL := 0.0;
    robot6axis/servo_2/servo_mode/offsetAxToMa1 AT 6706 : REAL := 0.0;
    robot6axis/servo_2/servo_mode/ActualPositionMa_o1 AT 6707 : REAL := 0.0;
    robot6axis/servo_2/servo_control/HomeCmd AT 70 : BOOL := false;
    robot6axis/servo_2/servo_control/MoveVelCmd AT 69 : BOOL := false;
    robot6axis/servo_2/servo_control/MoveAbsCmd AT 68 : BOOL := false;
    robot6axis/servo_2/servo_control/MoveVel1ManualCmd AT 67 : BOOL := false;
    robot6axis/servo_2/servo_control/MoveVel2ManualCmd AT 66 : BOOL := false;
    robot6axis/servo_2/servo_control/MoveAbs1ManualCmd AT 65 : BOOL := false;
    robot6axis/servo_2/servo_control/MoveAbs2ManualCmd AT 64 : BOOL := false;
    robot6axis/servo_2/servo_control/StopCmd AT 14 : BOOL := false;
    robot6axis/servo_2/servo_control/MovePosition AT 79 : REAL := 0.0;
    robot6axis/servo_2/servo_control/MoveSpeed AT 78 : REAL := 100.0;
    robot6axis/servo_2/servo_control/MoveAcceleration AT 77 : REAL := 100.0;
    robot6axis/servo_2/servo_control/MoveDeceleration AT 76 : REAL := 100.0;
    robot6axis/servo_2/servo_control/offsetAxToMa AT 75 : REAL := 0.0;
    robot6axis/servo_2/servo_control/physicalPosInit AT 6491 : REAL := 0.0;
    robot6axis/servo_2/servo_control/MAX_SPEED AT 6490 : REAL(0.0..3.4e+038) := 30.0;
    robot6axis/servo_2/servo_control/status AT 627 : INT := 0;
    robot6axis/servo_2/servo_control/errorFlag AT 626 : INT := 0;
    robot6axis/servo_2/servo_control/IOActualPositionAx AT 6493 : REAL := 0.0;
    robot6axis/servo_2/servo_control/IOVelDone AT 204 : BOOL := false;
    robot6axis/servo_2/servo_control/IOAbsDone AT 203 : BOOL := false;
    robot6axis/servo_2/servo_control/IOActualVelocity AT 6492 : REAL := 0.0;
    robot6axis/servo_2/servo_control/OperationMode AT 643 : INT := 0;
    robot6axis/servo_2/servo_control/StatusReady AT 232 : BOOL := true;
    robot6axis/servo_2/servo_control/StatusMove AT 233 : BOOL := false;
    robot6axis/servo_2/servo_control/StatusStand AT 234 : BOOL := false;
    robot6axis/servo_2/servo_control/ActualPositionMa AT 6694 : REAL := 0.0;
    robot6axis/servo_2/servo_control/ActualVelocity AT 6695 : REAL := 0.0;
    robot6axis/servo_2/servo_control/MaximumVelocity AT 6696 : REAL := 0.0;
    robot6axis/servo_2/servo_control/VelEnabled AT 235 : BOOL := false;
    robot6axis/servo_2/servo_control/VelCmd AT 236 : BOOL := false;
    robot6axis/servo_2/servo_control/PosEnabled AT 237 : BOOL := false;
    robot6axis/servo_2/servo_control/PosCmd AT 238 : BOOL := false;
    robot6axis/servo_2/servo_control/Position AT 6698 : REAL := 0.0;
    robot6axis/servo_2/servo_control/Speed AT 6697 : REAL := 0.0;
    robot6axis/servo_2/servo_control/ManualMode AT 644 : INT := 0;
    robot6axis/servo_2/servo_control/initDone AT 242 : BOOL := false;
    robot6axis/servo_2/servo_control/ActualPositionMa1 AT 6708 : REAL := 0.0;
    robot6axis/servo_2/servo_control/offsetAxToMa1 AT 6709 : REAL := 0.0;
    robot6axis/servo_2/servo_control/HOME_POSITION AT 6710 : REAL := 100.0;
    robot6axis/servo_2/servo_control/MANUAL_POSITION1 AT 6711 : REAL := 0.0;
    robot6axis/servo_2/servo_control/MANUAL_POSITION2 AT 6712 : REAL := 150.0;
    robot6axis/servo_2/servo_control/MANUAL_SPEED1 AT 6713 : REAL := -100.0;
    robot6axis/servo_2/servo_control/MANUAL_SPEED2 AT 6714 : REAL := 100.0;
    robot6axis/servo_2/servo_control/MANUAL_SPEED AT 6715 : REAL := 100.0;
    robot6axis/servo_2/servo_velocity/MoveVelEnable AT 235 : BOOL := false;
    robot6axis/servo_2/servo_velocity/MoveVelStart AT 236 : BOOL := false;
    robot6axis/servo_2/servo_velocity/MoveSpeed AT 6697 : REAL := 0.0;
    robot6axis/servo_2/servo_velocity/MoveAcceleration AT 77 : REAL := 100.0;
    robot6axis/servo_2/servo_velocity/MoveDeceleration AT 76 : REAL := 100.0;
    robot6axis/servo_2/servo_velocity/MAX_SPEED AT 6490 : REAL(0.0..3.4e+038) := 30.0;
    robot6axis/servo_2/servo_velocity/MAX_ACCEL AT 6489 : REAL(0.0..3.4e+038) := 1500.0;
    robot6axis/servo_2/servo_velocity/MAX_DECEL AT 6488 : REAL(0.0..3.4e+038) := 1500.0;
    robot6axis/servo_2/servo_velocity/MODULO_LENGTH AT 6487 : REAL := 0.0;
    robot6axis/servo_2/servo_velocity/status AT 627 : INT := 0;
    robot6axis/servo_2/servo_velocity/errorFlag AT 626 : INT := 0;
    robot6axis/servo_2/servo_velocity/MoveVelDone AT 204 : BOOL := false;
    robot6axis/servo_2/servo_velocity/ActualPositionAx AT 6493 : REAL := 0.0;
    robot6axis/servo_2/servo_velocity/ActualVelocity AT 6492 : REAL := 0.0;
    robot6axis/servo_2/servo_velocity/firstStep AT 243 : BOOL := true;
    robot6axis/servo_2/servo_velocity/stepDone AT 244 : BOOL := false;
    robot6axis/servo_2/servo_velocity/currentTime AT 6716 : REAL := 0.0;
    robot6axis/servo_2/servo_velocity/MoveSpeed1 AT 6717 : REAL := 0.0;
    robot6axis/servo_2/servo_velocity/acceleration AT 6718 : REAL := 0.0;
    robot6axis/servo_2/servo_velocity/deceleration AT 6719 : REAL := 0.0;
    robot6axis/servo_2/servo_velocity/orderSpeed AT 6720 : REAL := 0.0;
    robot6axis/servo_2/servo_velocity/endChangeSpeed AT 6721 : REAL := 0.0;
    robot6axis/servo_2/servo_velocity/accelDecelChangeSpeed AT 6722 : REAL := 0.0;
    robot6axis/servo_2/servo_velocity/ActualVelocity1 AT 6723 : REAL := 0.0;
    robot6axis/servo_2/servo_velocity/speedChanged AT 245 : BOOL := false;
    robot6axis/servo_2/servo_position/MoveAbsEnable AT 237 : BOOL := false;
    robot6axis/servo_2/servo_position/MoveAbsStart AT 238 : BOOL := false;
    robot6axis/servo_2/servo_position/MovePosition AT 6698 : REAL := 0.0;
    robot6axis/servo_2/servo_position/MoveSpeed AT 6697 : REAL := 0.0;
    robot6axis/servo_2/servo_position/MoveAcceleration AT 77 : REAL := 100.0;
    robot6axis/servo_2/servo_position/MoveDeceleration AT 76 : REAL := 100.0;
    robot6axis/servo_2/servo_position/MAX_SPEED AT 6490 : REAL(0.0..3.4e+038) := 30.0;
    robot6axis/servo_2/servo_position/MAX_ACCEL AT 6489 : REAL(0.0..3.4e+038) := 1500.0;
    robot6axis/servo_2/servo_position/MAX_DECEL AT 6488 : REAL(0.0..3.4e+038) := 1500.0;
    robot6axis/servo_2/servo_position/MODULO_LENGTH AT 6487 : REAL := 0.0;
    robot6axis/servo_2/servo_position/status AT 627 : INT := 0;
    robot6axis/servo_2/servo_position/errorFlag AT 626 : INT := 0;
    robot6axis/servo_2/servo_position/MoveAbsDone AT 203 : BOOL := false;
    robot6axis/servo_2/servo_position/ActualPositionAx AT 6493 : REAL := 0.0;
    robot6axis/servo_2/servo_position/ActualVelocity AT 6492 : REAL := 0.0;
    robot6axis/servo_2/servo_position/firstStep AT 246 : BOOL := true;
    robot6axis/servo_2/servo_position/stepDone AT 247 : BOOL := false;
    robot6axis/servo_2/servo_position/timeToStop AT 6724 : REAL := 0.0;
    robot6axis/servo_2/servo_position/distanceToStop AT 6725 : REAL := 0.0;
    robot6axis/servo_2/servo_position/distance AT 6726 : REAL := 0.0;
    robot6axis/servo_2/servo_position/currentTime AT 6727 : REAL := 0.0;
    robot6axis/servo_2/servo_position/currentSpeed1 AT 6728 : REAL := 0.0;
    robot6axis/servo_2/servo_position/targetPosition AT 6729 : REAL := 0.0;
    robot6axis/servo_2/servo_position/ActualPositionAx1 AT 6730 : REAL := 0.0;
    robot6axis/servo_2/servo_position/acceleration AT 6731 : REAL := 0.0;
    robot6axis/servo_2/servo_position/deceleration AT 6732 : REAL := 0.0;
    robot6axis/servo_2/servo_position/orderSpeed AT 6733 : REAL := 0.0;
    robot6axis/servo_2/servo_position/moveDirection AT 6734 : REAL := 0.0;
    robot6axis/servo_2/servo_position/moveDirection1 AT 6735 : REAL := 0.0;
    robot6axis/servo_2/servo_position/endChangeSpeed AT 6736 : REAL := 0.0;
    robot6axis/servo_2/servo_position/ActualVelocity1 AT 6737 : REAL := 0.0;
    robot6axis/arm2/armOrigin AT 6531 : ARRAY[1..3] OF REAL := [3(0.0)];
    robot6axis/arm2/overallArmQuatInput AT 6536 : ARRAY[1..4] OF REAL := [4(0.0)];
    robot6axis/arm2/structRotVector AT 140 : ARRAY[1..3] OF REAL := [2(0.0), 1.0];
    robot6axis/arm2/structRotDeg AT 139 : REAL := -90.0;
    robot6axis/arm2/driveRotVector AT 129 : ARRAY[1..3] OF REAL := [0.0, 1.0, 0.0];
    robot6axis/arm2/driveRotDeg AT 6542 : REAL := 0.0;
    robot6axis/arm2/ownRotDeg AT 6483 : REAL := 0.0;
    robot6axis/arm2/driveResizeLength AT 6482 : REAL := 0.0;
    robot6axis/arm2/functionActive AT 197 : BOOL := false;
    robot6axis/arm2/armExtrem AT 6543 : ARRAY[1..3] OF REAL := [3(0.0)];
    robot6axis/arm2/overallArmRotOutput AT 6548 : ARRAY[1..4] OF REAL := [4(0.0)];
    robot6axis/arm2/productId AT 625 : DINT := -1;
    robot6axis/arm2/status_act_prod AT 645 : DINT := 0;
    robot6axis/arm2/m11 AT 6738 : REAL := 50.9284;
    robot6axis/arm2/m12 AT 6739 : REAL := 0.0;
    robot6axis/arm2/m13 AT 6740 : REAL := 0.0;
    robot6axis/arm2/m14 AT 6741 : REAL := 16.9761;
    robot6axis/arm2/m21 AT 6742 : REAL := 0.0;
    robot6axis/arm2/m22 AT 6743 : REAL := 32.1839;
    robot6axis/arm2/m23 AT 6744 : REAL := 0.0;
    robot6axis/arm2/m24 AT 6745 : REAL := 96.1981;
    robot6axis/arm2/m31 AT 6746 : REAL := 0.0;
    robot6axis/arm2/m32 AT 6747 : REAL := 0.0;
    robot6axis/arm2/m33 AT 6748 : REAL := 12.7321;
    robot6axis/arm2/m34 AT 6749 : REAL := 53.0504;
    robot6axis/arm2/m41 AT 6750 : REAL := 0.0;
    robot6axis/arm2/m42 AT 6751 : REAL := 0.0;
    robot6axis/arm2/m43 AT 6752 : REAL := 0.0;
    robot6axis/arm2/m44 AT 6753 : REAL := 1.0;
    robot6axis/arm2/armLengthCalc AT 6754 : REAL := 0.0;
    robot6axis/arm2/functionActiveLocale AT 248 : BOOL := false;
    robot6axis/arm2/product_id AT 646 : DINT := -1;
    robot6axis/arm2/arm_id AT 647 : DINT := -1;
    robot6axis/arm2/timeToGripParam AT 6755 : REAL := 0.15;
    robot6axis/arm2/armLength AT 6756 : REAL := 290.0;
    robot6axis/arm2/armWidth AT 6757 : REAL := 60.0;
    robot6axis/arm2/armHeight AT 6758 : REAL := 60.0;
    robot6axis/arm2/armType AT 648 : INT := 0;
    robot6axis/servo_3/status AT 624 : INT := 0;
    robot6axis/servo_3/errorFlag AT 623 : INT := 0;
    robot6axis/servo_3/ActualPositionAx1 AT 6481 : REAL := 0.0;
    robot6axis/servo_3/MoveVelDone1 AT 196 : BOOL := false;
    robot6axis/servo_3/ActualVelocity1 AT 6480 : REAL := 0.0;
    robot6axis/servo_3/MoveAbsDone1 AT 195 : BOOL := false;
    robot6axis/servo_3/HomeCmd AT 63 : BOOL := false;
    robot6axis/servo_3/MoveVelCmd AT 62 : BOOL := false;
    robot6axis/servo_3/MoveAbsCmd AT 61 : BOOL := false;
    robot6axis/servo_3/MoveVel1ManualCmd AT 60 : BOOL := false;
    robot6axis/servo_3/MoveVel2ManualCmd AT 59 : BOOL := false;
    robot6axis/servo_3/MoveAbs1ManualCmd AT 58 : BOOL := false;
    robot6axis/servo_3/MoveAbs2ManualCmd AT 57 : BOOL := false;
    robot6axis/servo_3/StopCmd AT 14 : BOOL := false;
    robot6axis/servo_3/MovePosition AT 74 : REAL := 0.0;
    robot6axis/servo_3/MoveSpeed AT 73 : REAL := 100.0;
    robot6axis/servo_3/MoveAcceleration AT 72 : REAL := 100.0;
    robot6axis/servo_3/MoveDeceleration AT 71 : REAL := 100.0;
    robot6axis/servo_3/offsetAxToMa AT 70 : REAL := 0.0;
    robot6axis/servo_3/PLC_StatusReady AT 29 : BOOL := true;
    robot6axis/servo_3/PLC_StatusMoved AT 28 : BOOL := false;
    robot6axis/servo_3/PLC_StatusStand AT 27 : BOOL := false;
    robot6axis/servo_3/PLC_ActualPositionAx AT 160 : REAL := 0.0;
    robot6axis/servo_3/PLC_ActualPositionMa AT 50 : REAL := 0.0;
    robot6axis/servo_3/PLC_ActualVelocity AT 49 : REAL := 0.0;
    robot6axis/servo_3/physicalPosInit AT 6479 : REAL := 0.0;
    robot6axis/servo_3/MAX_SPEED AT 6478 : REAL(0.0..3.4e+038) := 30.0;
    robot6axis/servo_3/MAX_ACCEL AT 6477 : REAL(0.0..3.4e+038) := 1500.0;
    robot6axis/servo_3/MAX_DECEL AT 6476 : REAL(0.0..3.4e+038) := 1500.0;
    robot6axis/servo_3/MODULO_LENGTH AT 6475 : REAL := 0.0;
    robot6axis/servo_3/StatusReady AT 194 : BOOL := true;
    robot6axis/servo_3/StatusMoved AT 193 : BOOL := false;
    robot6axis/servo_3/StatusStand AT 192 : BOOL := false;
    robot6axis/servo_3/ActualPositionAx AT 6554 : REAL := 0.0;
    robot6axis/servo_3/ActualPositionMa AT 6474 : REAL := 0.0;
    robot6axis/servo_3/ActualVelocity AT 40 : REAL := 0.0;
    robot6axis/servo_3/MaximumVelocity AT 6473 : REAL := 0.0;
    robot6axis/servo_3/StatusPosIncrease AT 191 : BOOL := false;
    robot6axis/servo_3/StatusPosDecrease AT 190 : BOOL := false;
    robot6axis/servo_3/displayJauge AT 6472 : REAL := 0.0;
    robot6axis/servo_3/servo_mode/PLC_StatusReady AT 29 : BOOL := true;
    robot6axis/servo_3/servo_mode/PLC_StatusMoved AT 28 : BOOL := false;
    robot6axis/servo_3/servo_mode/PLC_StatusStand AT 27 : BOOL := false;
    robot6axis/servo_3/servo_mode/PLC_ActualPositionAx AT 160 : REAL := 0.0;
    robot6axis/servo_3/servo_mode/PLC_ActualPositionMa AT 50 : REAL := 0.0;
    robot6axis/servo_3/servo_mode/PLC_ActualVelocity AT 49 : REAL := 0.0;
    robot6axis/servo_3/servo_mode/StatusReady AT 249 : BOOL := true;
    robot6axis/servo_3/servo_mode/StatusMoved AT 250 : BOOL := false;
    robot6axis/servo_3/servo_mode/StatusStand AT 251 : BOOL := false;
    robot6axis/servo_3/servo_mode/ActualPositionMa AT 6759 : REAL := 0.0;
    robot6axis/servo_3/servo_mode/ActualVelocity AT 6760 : REAL := 0.0;
    robot6axis/servo_3/servo_mode/MaximumVelocity AT 6761 : REAL := 0.0;
    robot6axis/servo_3/servo_mode/physicalPosInit AT 6479 : REAL := 0.0;
    robot6axis/servo_3/servo_mode/ActualPositionAx AT 6481 : REAL := 0.0;
    robot6axis/servo_3/servo_mode/StatusReady_o AT 194 : BOOL := true;
    robot6axis/servo_3/servo_mode/StatusMoved_o AT 193 : BOOL := false;
    robot6axis/servo_3/servo_mode/StatusStand_o AT 192 : BOOL := false;
    robot6axis/servo_3/servo_mode/ActualPositionAx_o AT 6554 : REAL := 0.0;
    robot6axis/servo_3/servo_mode/ActualPositionMa_o AT 6474 : REAL := 0.0;
    robot6axis/servo_3/servo_mode/ActualVelocity_o AT 40 : REAL := 0.0;
    robot6axis/servo_3/servo_mode/MaximumVelocity_o AT 6473 : REAL := 0.0;
    robot6axis/servo_3/servo_mode/StatusPosIncrease_o AT 191 : BOOL := false;
    robot6axis/servo_3/servo_mode/StatusPosDecrease_o AT 190 : BOOL := false;
    robot6axis/servo_3/servo_mode/displayJauge_o AT 6472 : REAL := 0.0;
    robot6axis/servo_3/servo_mode/PLCMode AT 256 : BOOL := false;
    robot6axis/servo_3/servo_mode/PLCMode1 AT 257 : BOOL := false;
    robot6axis/servo_3/servo_mode/initDone AT 258 : BOOL := false;
    robot6axis/servo_3/servo_mode/displayPosMin AT 6764 : REAL := 0.0;
    robot6axis/servo_3/servo_mode/displayPosMax AT 6765 : REAL := 0.0;
    robot6axis/servo_3/servo_mode/PLC_ActualPositionAx1 AT 6766 : REAL := 0.0;
    robot6axis/servo_3/servo_mode/PLC_ActualVelocity1 AT 6767 : REAL := 0.0;
    robot6axis/servo_3/servo_mode/ActualPositionAx1 AT 6768 : REAL := 0.0;
    robot6axis/servo_3/servo_mode/ActualVelocity1 AT 6769 : REAL := 0.0;
    robot6axis/servo_3/servo_mode/offsetAxToMa AT 6770 : REAL := 0.0;
    robot6axis/servo_3/servo_mode/offsetAxToMa1 AT 6771 : REAL := 0.0;
    robot6axis/servo_3/servo_mode/ActualPositionMa_o1 AT 6772 : REAL := 0.0;
    robot6axis/servo_3/servo_control/HomeCmd AT 63 : BOOL := false;
    robot6axis/servo_3/servo_control/MoveVelCmd AT 62 : BOOL := false;
    robot6axis/servo_3/servo_control/MoveAbsCmd AT 61 : BOOL := false;
    robot6axis/servo_3/servo_control/MoveVel1ManualCmd AT 60 : BOOL := false;
    robot6axis/servo_3/servo_control/MoveVel2ManualCmd AT 59 : BOOL := false;
    robot6axis/servo_3/servo_control/MoveAbs1ManualCmd AT 58 : BOOL := false;
    robot6axis/servo_3/servo_control/MoveAbs2ManualCmd AT 57 : BOOL := false;
    robot6axis/servo_3/servo_control/StopCmd AT 14 : BOOL := false;
    robot6axis/servo_3/servo_control/MovePosition AT 74 : REAL := 0.0;
    robot6axis/servo_3/servo_control/MoveSpeed AT 73 : REAL := 100.0;
    robot6axis/servo_3/servo_control/MoveAcceleration AT 72 : REAL := 100.0;
    robot6axis/servo_3/servo_control/MoveDeceleration AT 71 : REAL := 100.0;
    robot6axis/servo_3/servo_control/offsetAxToMa AT 70 : REAL := 0.0;
    robot6axis/servo_3/servo_control/physicalPosInit AT 6479 : REAL := 0.0;
    robot6axis/servo_3/servo_control/MAX_SPEED AT 6478 : REAL(0.0..3.4e+038) := 30.0;
    robot6axis/servo_3/servo_control/status AT 624 : INT := 0;
    robot6axis/servo_3/servo_control/errorFlag AT 623 : INT := 0;
    robot6axis/servo_3/servo_control/IOActualPositionAx AT 6481 : REAL := 0.0;
    robot6axis/servo_3/servo_control/IOVelDone AT 196 : BOOL := false;
    robot6axis/servo_3/servo_control/IOAbsDone AT 195 : BOOL := false;
    robot6axis/servo_3/servo_control/IOActualVelocity AT 6480 : REAL := 0.0;
    robot6axis/servo_3/servo_control/OperationMode AT 649 : INT := 0;
    robot6axis/servo_3/servo_control/StatusReady AT 249 : BOOL := true;
    robot6axis/servo_3/servo_control/StatusMove AT 250 : BOOL := false;
    robot6axis/servo_3/servo_control/StatusStand AT 251 : BOOL := false;
    robot6axis/servo_3/servo_control/ActualPositionMa AT 6759 : REAL := 0.0;
    robot6axis/servo_3/servo_control/ActualVelocity AT 6760 : REAL := 0.0;
    robot6axis/servo_3/servo_control/MaximumVelocity AT 6761 : REAL := 0.0;
    robot6axis/servo_3/servo_control/VelEnabled AT 252 : BOOL := false;
    robot6axis/servo_3/servo_control/VelCmd AT 253 : BOOL := false;
    robot6axis/servo_3/servo_control/PosEnabled AT 254 : BOOL := false;
    robot6axis/servo_3/servo_control/PosCmd AT 255 : BOOL := false;
    robot6axis/servo_3/servo_control/Position AT 6763 : REAL := 0.0;
    robot6axis/servo_3/servo_control/Speed AT 6762 : REAL := 0.0;
    robot6axis/servo_3/servo_control/ManualMode AT 650 : INT := 0;
    robot6axis/servo_3/servo_control/initDone AT 259 : BOOL := false;
    robot6axis/servo_3/servo_control/ActualPositionMa1 AT 6773 : REAL := 0.0;
    robot6axis/servo_3/servo_control/offsetAxToMa1 AT 6774 : REAL := 0.0;
    robot6axis/servo_3/servo_control/HOME_POSITION AT 6775 : REAL := 100.0;
    robot6axis/servo_3/servo_control/MANUAL_POSITION1 AT 6776 : REAL := 0.0;
    robot6axis/servo_3/servo_control/MANUAL_POSITION2 AT 6777 : REAL := 150.0;
    robot6axis/servo_3/servo_control/MANUAL_SPEED1 AT 6778 : REAL := -100.0;
    robot6axis/servo_3/servo_control/MANUAL_SPEED2 AT 6779 : REAL := 100.0;
    robot6axis/servo_3/servo_control/MANUAL_SPEED AT 6780 : REAL := 100.0;
    robot6axis/servo_3/servo_velocity/MoveVelEnable AT 252 : BOOL := false;
    robot6axis/servo_3/servo_velocity/MoveVelStart AT 253 : BOOL := false;
    robot6axis/servo_3/servo_velocity/MoveSpeed AT 6762 : REAL := 0.0;
    robot6axis/servo_3/servo_velocity/MoveAcceleration AT 72 : REAL := 100.0;
    robot6axis/servo_3/servo_velocity/MoveDeceleration AT 71 : REAL := 100.0;
    robot6axis/servo_3/servo_velocity/MAX_SPEED AT 6478 : REAL(0.0..3.4e+038) := 30.0;
    robot6axis/servo_3/servo_velocity/MAX_ACCEL AT 6477 : REAL(0.0..3.4e+038) := 1500.0;
    robot6axis/servo_3/servo_velocity/MAX_DECEL AT 6476 : REAL(0.0..3.4e+038) := 1500.0;
    robot6axis/servo_3/servo_velocity/MODULO_LENGTH AT 6475 : REAL := 0.0;
    robot6axis/servo_3/servo_velocity/status AT 624 : INT := 0;
    robot6axis/servo_3/servo_velocity/errorFlag AT 623 : INT := 0;
    robot6axis/servo_3/servo_velocity/MoveVelDone AT 196 : BOOL := false;
    robot6axis/servo_3/servo_velocity/ActualPositionAx AT 6481 : REAL := 0.0;
    robot6axis/servo_3/servo_velocity/ActualVelocity AT 6480 : REAL := 0.0;
    robot6axis/servo_3/servo_velocity/firstStep AT 260 : BOOL := true;
    robot6axis/servo_3/servo_velocity/stepDone AT 261 : BOOL := false;
    robot6axis/servo_3/servo_velocity/currentTime AT 6781 : REAL := 0.0;
    robot6axis/servo_3/servo_velocity/MoveSpeed1 AT 6782 : REAL := 0.0;
    robot6axis/servo_3/servo_velocity/acceleration AT 6783 : REAL := 0.0;
    robot6axis/servo_3/servo_velocity/deceleration AT 6784 : REAL := 0.0;
    robot6axis/servo_3/servo_velocity/orderSpeed AT 6785 : REAL := 0.0;
    robot6axis/servo_3/servo_velocity/endChangeSpeed AT 6786 : REAL := 0.0;
    robot6axis/servo_3/servo_velocity/accelDecelChangeSpeed AT 6787 : REAL := 0.0;
    robot6axis/servo_3/servo_velocity/ActualVelocity1 AT 6788 : REAL := 0.0;
    robot6axis/servo_3/servo_velocity/speedChanged AT 262 : BOOL := false;
    robot6axis/servo_3/servo_position/MoveAbsEnable AT 254 : BOOL := false;
    robot6axis/servo_3/servo_position/MoveAbsStart AT 255 : BOOL := false;
    robot6axis/servo_3/servo_position/MovePosition AT 6763 : REAL := 0.0;
    robot6axis/servo_3/servo_position/MoveSpeed AT 6762 : REAL := 0.0;
    robot6axis/servo_3/servo_position/MoveAcceleration AT 72 : REAL := 100.0;
    robot6axis/servo_3/servo_position/MoveDeceleration AT 71 : REAL := 100.0;
    robot6axis/servo_3/servo_position/MAX_SPEED AT 6478 : REAL(0.0..3.4e+038) := 30.0;
    robot6axis/servo_3/servo_position/MAX_ACCEL AT 6477 : REAL(0.0..3.4e+038) := 1500.0;
    robot6axis/servo_3/servo_position/MAX_DECEL AT 6476 : REAL(0.0..3.4e+038) := 1500.0;
    robot6axis/servo_3/servo_position/MODULO_LENGTH AT 6475 : REAL := 0.0;
    robot6axis/servo_3/servo_position/status AT 624 : INT := 0;
    robot6axis/servo_3/servo_position/errorFlag AT 623 : INT := 0;
    robot6axis/servo_3/servo_position/MoveAbsDone AT 195 : BOOL := false;
    robot6axis/servo_3/servo_position/ActualPositionAx AT 6481 : REAL := 0.0;
    robot6axis/servo_3/servo_position/ActualVelocity AT 6480 : REAL := 0.0;
    robot6axis/servo_3/servo_position/firstStep AT 263 : BOOL := true;
    robot6axis/servo_3/servo_position/stepDone AT 264 : BOOL := false;
    robot6axis/servo_3/servo_position/timeToStop AT 6789 : REAL := 0.0;
    robot6axis/servo_3/servo_position/distanceToStop AT 6790 : REAL := 0.0;
    robot6axis/servo_3/servo_position/distance AT 6791 : REAL := 0.0;
    robot6axis/servo_3/servo_position/currentTime AT 6792 : REAL := 0.0;
    robot6axis/servo_3/servo_position/currentSpeed1 AT 6793 : REAL := 0.0;
    robot6axis/servo_3/servo_position/targetPosition AT 6794 : REAL := 0.0;
    robot6axis/servo_3/servo_position/ActualPositionAx1 AT 6795 : REAL := 0.0;
    robot6axis/servo_3/servo_position/acceleration AT 6796 : REAL := 0.0;
    robot6axis/servo_3/servo_position/deceleration AT 6797 : REAL := 0.0;
    robot6axis/servo_3/servo_position/orderSpeed AT 6798 : REAL := 0.0;
    robot6axis/servo_3/servo_position/moveDirection AT 6799 : REAL := 0.0;
    robot6axis/servo_3/servo_position/moveDirection1 AT 6800 : REAL := 0.0;
    robot6axis/servo_3/servo_position/endChangeSpeed AT 6801 : REAL := 0.0;
    robot6axis/servo_3/servo_position/ActualVelocity1 AT 6802 : REAL := 0.0;
    robot6axis/arm3/armOrigin AT 6543 : ARRAY[1..3] OF REAL := [3(0.0)];
    robot6axis/arm3/overallArmQuatInput AT 6548 : ARRAY[1..4] OF REAL := [4(0.0)];
    robot6axis/arm3/structRotVector AT 6467 : ARRAY[1..3] OF REAL := [2(0.0), 1.0];
    robot6axis/arm3/structRotDeg AT 6466 : REAL := 0.0;
    robot6axis/arm3/driveRotVector AT 124 : ARRAY[1..3] OF REAL := [0.0, 1.0, 0.0];
    robot6axis/arm3/driveRotDeg AT 6554 : REAL := 0.0;
    robot6axis/arm3/ownRotDeg AT 6465 : REAL := 0.0;
    robot6axis/arm3/driveResizeLength AT 6464 : REAL := 0.0;
    robot6axis/arm3/functionActive AT 189 : BOOL := false;
    robot6axis/arm3/armExtrem AT 6555 : ARRAY[1..3] OF REAL := [3(0.0)];
    robot6axis/arm3/overallArmRotOutput AT 6560 : ARRAY[1..4] OF REAL := [4(0.0)];
    robot6axis/arm3/productId AT 622 : DINT := -1;
    robot6axis/arm3/status_act_prod AT 651 : DINT := 0;
    robot6axis/arm3/m11 AT 6803 : REAL := 43.855;
    robot6axis/arm3/m12 AT 6804 : REAL := 0.0;
    robot6axis/arm3/m13 AT 6805 : REAL := 0.0;
    robot6axis/arm3/m14 AT 6806 : REAL := 19.8055;
    robot6axis/arm3/m21 AT 6807 : REAL := 0.0;
    robot6axis/arm3/m22 AT 6808 : REAL := 32.1839;
    robot6axis/arm3/m23 AT 6809 : REAL := 0.0;
    robot6axis/arm3/m24 AT 6810 : REAL := 96.1981;
    robot6axis/arm3/m31 AT 6811 : REAL := 0.0;
    robot6axis/arm3/m32 AT 6812 : REAL := 0.0;
    robot6axis/arm3/m33 AT 6813 : REAL := 15.5615;
    robot6axis/arm3/m34 AT 6814 : REAL := 31.8302;
    robot6axis/arm3/m41 AT 6815 : REAL := 0.0;
    robot6axis/arm3/m42 AT 6816 : REAL := 0.0;
    robot6axis/arm3/m43 AT 6817 : REAL := 0.0;
    robot6axis/arm3/m44 AT 6818 : REAL := 1.0;
    robot6axis/arm3/armLengthCalc AT 6819 : REAL := 0.0;
    robot6axis/arm3/functionActiveLocale AT 265 : BOOL := false;
    robot6axis/arm3/product_id AT 652 : DINT := -1;
    robot6axis/arm3/arm_id AT 653 : DINT := -1;
    robot6axis/arm3/timeToGripParam AT 6820 : REAL := 0.15;
    robot6axis/arm3/armLength AT 6821 : REAL := 108.0;
    robot6axis/arm3/armWidth AT 6822 : REAL := 60.0;
    robot6axis/arm3/armHeight AT 6823 : REAL := 60.0;
    robot6axis/arm3/armType AT 654 : INT := 0;
    robot6axis/servo_4/status AT 621 : INT := 0;
    robot6axis/servo_4/errorFlag AT 620 : INT := 0;
    robot6axis/servo_4/ActualPositionAx1 AT 6463 : REAL := 0.0;
    robot6axis/servo_4/MoveVelDone1 AT 188 : BOOL := false;
    robot6axis/servo_4/ActualVelocity1 AT 6462 : REAL := 0.0;
    robot6axis/servo_4/MoveAbsDone1 AT 187 : BOOL := false;
    robot6axis/servo_4/HomeCmd AT 56 : BOOL := false;
    robot6axis/servo_4/MoveVelCmd AT 55 : BOOL := false;
    robot6axis/servo_4/MoveAbsCmd AT 54 : BOOL := false;
    robot6axis/servo_4/MoveVel1ManualCmd AT 53 : BOOL := false;
    robot6axis/servo_4/MoveVel2ManualCmd AT 52 : BOOL := false;
    robot6axis/servo_4/MoveAbs1ManualCmd AT 51 : BOOL := false;
    robot6axis/servo_4/MoveAbs2ManualCmd AT 50 : BOOL := false;
    robot6axis/servo_4/StopCmd AT 14 : BOOL := false;
    robot6axis/servo_4/MovePosition AT 69 : REAL := 0.0;
    robot6axis/servo_4/MoveSpeed AT 68 : REAL := 100.0;
    robot6axis/servo_4/MoveAcceleration AT 67 : REAL := 100.0;
    robot6axis/servo_4/MoveDeceleration AT 66 : REAL := 100.0;
    robot6axis/servo_4/offsetAxToMa AT 65 : REAL := 0.0;
    robot6axis/servo_4/PLC_StatusReady AT 26 : BOOL := true;
    robot6axis/servo_4/PLC_StatusMoved AT 25 : BOOL := false;
    robot6axis/servo_4/PLC_StatusStand AT 24 : BOOL := false;
    robot6axis/servo_4/PLC_ActualPositionAx AT 161 : REAL := 0.0;
    robot6axis/servo_4/PLC_ActualPositionMa AT 48 : REAL := 0.0;
    robot6axis/servo_4/PLC_ActualVelocity AT 47 : REAL := 0.0;
    robot6axis/servo_4/physicalPosInit AT 6461 : REAL := 0.0;
    robot6axis/servo_4/MAX_SPEED AT 6460 : REAL(0.0..3.4e+038) := 30.0;
    robot6axis/servo_4/MAX_ACCEL AT 6459 : REAL(0.0..3.4e+038) := 1500.0;
    robot6axis/servo_4/MAX_DECEL AT 6458 : REAL(0.0..3.4e+038) := 1500.0;
    robot6axis/servo_4/MODULO_LENGTH AT 6457 : REAL := 0.0;
    robot6axis/servo_4/StatusReady AT 186 : BOOL := true;
    robot6axis/servo_4/StatusMoved AT 185 : BOOL := false;
    robot6axis/servo_4/StatusStand AT 184 : BOOL := false;
    robot6axis/servo_4/ActualPositionAx AT 6566 : REAL := 0.0;
    robot6axis/servo_4/ActualPositionMa AT 6456 : REAL := 0.0;
    robot6axis/servo_4/ActualVelocity AT 39 : REAL := 0.0;
    robot6axis/servo_4/MaximumVelocity AT 6455 : REAL := 0.0;
    robot6axis/servo_4/StatusPosIncrease AT 183 : BOOL := false;
